                                    
    SEAL_SEPARATE_STATES.Fault :
END_CASE


CASE releaseAndFeedSubState OF
    RELEASE_FEED_STATES.Idle :                        //
                                                        
    RELEASE_FEED_STATES.MoveJawOutAndDropBag :        // 
                                                    IF (motorizedSealFlatteners.state = SEAL_FLATTENER_STATES.MovedFlattenersOut OR NOT motorizedSealFlatteners.enable) 
                                                        AND (pressureBar.clamped OR NOT pressureBar.enable)
                                                        AND ((bagDelivery.state = BAG_DELIVERY_STATES.ReverseDone) OR Globals.enableDryCycle)
                                                        OR (bagDelivery.state =  BAG_DELIVERY_STATES.WaitingForPrinter AND zebraPrinter.enable)
                                                        OR NOT bagDelivery.enable
                                                        THEN
                                                            IF motorizedSealFlatteners.enable THEN
                                                                motorizedSealFlatteners.AutoMoveToClearance();
                                                            END_IF
                                                            
                                                            IF enableBagOpen THEN
                                                                pressureBar.OpenJawForBagFeed();
															ELSE
																pressureBar.OpenJaw();
                                                            END_IF
                                                            //IBD.OpenFull();
// 															IF enableBagOpen THEN
// 																bagOpenFingers.Release();
// 															END_IF
															
															IF enableIBDEject THEN
																IBD.CloseIBD();
															END_IF
															
															IF enableLoadPlate THEN
																rearLoadPlateRetract.Trigger();
															END_IF
															
															IF TO_DINT(HMIData.exitConveyorDwell) <> 0 THEN
																exitConveyorRun.Trigger();
															END_IF
															
															IF TO_DINT(HMIData.externalExitConveyorDwell) <> 0 THEN
																externalExitConveyorRun.Trigger();
															END_IF
															
															IF enableLabelSideUp THEN
																forwardLoadPlateRetract.Trigger();
																loadShelfExtend.Trigger();
															END_IF
															
															IF HMIData.lpaBagEjectAssistEnable THEN
																LPA.ManualOn();
															END_IF
															IBD.OpenFull();
                                                           bagDropTimer.IN := TRUE;
														   releaseAndFeedSubState := RELEASE_FEED_STATES.MovingJawOutAndDroppingBag;
                                                    END_IF
													
	 RELEASE_FEED_STATES.MovingJawOutAndDroppingBag :
														 // If printer is enabled then perform printer operation of bag delivery, otherwise just feed new bag out.
                                                            // In the case that bagDelivery is disabled then we're done with release and feed
														IF enableBagOpen AND pressureBar.actualPosition >= 0.5 THEN
 															bagOpenFingers.Release();
 														END_IF	
														
                                                        IF bagDropTimer.Q 
															AND (motorizedSealFlatteners.state = SEAL_FLATTENER_STATES.MovedFlattenersToBagFeed OR NOT motorizedSealFlatteners.enable)
															THEN   
															bagDropTimer.IN := FALSE;
															
															IF bagDelivery.enable AND NOT zebraPrinter.enable THEN
                                                                bagDelivery.AutoFeedBagOut();
																LPA.ManualOff();
																IF HMIData.lpaDuringBagFeedEnable THEN
																	LPA.ManualOn();
																END_IF
                                                                releaseAndFeedSubState := RELEASE_FEED_STATES.MovingJawOutAndFeedingBag;
                                                            ELSIF bagDelivery.enable AND zebraPrinter.enable THEN
                                                                bagDelivery.AutoWaitForPrinter();
																LPA.ManualOff();
                                                                releaseAndFeedSubState := RELEASE_FEED_STATES.WaitForPrinter;
                                                            ELSE 
                                                                releaseAndFeedSubState := RELEASE_FEED_STATES.Done;
                                                            END_IF
                                                            (*{warning 'TODO: This is a hack to use HPA as LPA'}
														    HPA.DwellSetting := 500;		// Get rid on this - ha
													        HPA.Trigger();*)												
    													END_IF
														
    RELEASE_FEED_STATES.WaitForPrinter :            // Data Ready means the printer has a label and we're all set to print
                                                    IF zebraPrinter.state = PRINTER_STATES.DataReady THEN
                                                        releaseAndFeedSubState := RELEASE_FEED_STATES.FeedToOffset;
                                                    END_IF
                                                    
    RELEASE_FEED_STATES.FeedToOffset :              // This starts feeding to the print offset
													IF (motorizedSealFlatteners.state = SEAL_FLATTENER_STATES.MovedFlattenersToBagFeed OR NOT motorizedSealFlatteners.enable) THEN
														bagDelivery.AutoPrinterReady();
                                                    	releaseAndFeedSubState := RELEASE_FEED_STATES.FeedingToOffset;
													END_IF
                                                    
                                                        
    RELEASE_FEED_STATES.FeedingToOffset :            // Once offset done start printing
                                                    IF bagDelivery.state = BAG_DELIVERY_STATES.FedToPrintOffset THEN
                                                        releaseAndFeedSubState := RELEASE_FEED_STATES.StartPrinting;
                                                    END_IF                                            
    
    RELEASE_FEED_STATES.StartPrinting :                // Printer starts print cycle and bag delivery starts moving at print speed
                                                    
                                                    //bagDelivery.AutoStartPrintFeed();
													zebraPrinter.AutoPrintNow();
                                                    
                                                    releaseAndFeedSubState := RELEASE_FEED_STATES.SendPrintSignal;                                            

    RELEASE_FEED_STATES.SendPrintSignal:            // 
                                                    //IF bagDelivery.state =     BAG_DELIVERY_STATES.FeedingAtPrintSpeed THEN
													//zebraPrinter.AutoSendPrintSignal();
													IF zebraPrinter.printHeadDebounced THEN
														bagDelivery.AutoStartPrintFeed();
														zebraPrinter.AutoSendPrintSignal();
														barcodeVerifier.Trigger();
                                                        //bagDelivery.AutoStartPrintFeed();
														//bagDelivery.AutoStartPrintFeed();
                                                        //zebraPrinter.AutoSendPrintSignal();
														
                                                        releaseAndFeedSubState := RELEASE_FEED_STATES.Printing;
                                                    END_IF                                        

    RELEASE_FEED_STATES.Printing :                // 
													
                                                    IF zebraPrinter.state = PRINTER_STATES.DonePrinting THEN
                                                        releaseAndFeedSubState := RELEASE_FEED_STATES.StopPrinting;
                                                    END_IF
                                                    
    RELEASE_FEED_STATES.StopPrinting :                // Tell bag delivery it's okay to feed out the rest of the bag and the printer that it can prep itself for the next print
                                                    bagDelivery.AutoPrinterDone();
                                                    zebraPrinter.AutoAckPrintDone();
													IF HMIData.lpaDuringBagFeedEnable THEN
														LPA.ManualOn();
													END_IF
													
                                                    releaseAndFeedSubState := RELEASE_FEED_STATES.MovingJawOutAndFeedingBag;
                                                                                
                                                                                                            
    RELEASE_FEED_STATES.MovingJawOutAndFeedingBag :    // 
    
													
													IF (bagdelivery.state = BAG_DELIVERY_STATES.Ready OR NOT bagdelivery.enable)
                                                        AND (motorizedSealFlatteners.state = SEAL_FLATTENER_STATES.MovedFlattenersToBagFeed OR NOT motorizedSealFlatteners.enable) 
                                                        AND (pressureBar.pressureBarOpen OR NOT pressureBar.enable)
                                                        THEN
															IF LPA.DwellSetting = 0 THEN
																LPA.ManualOff();
															END_IF
															//IBD.OpenIBD();
                                                            releaseAndFeedSubState := RELEASE_FEED_STATES.MovedJawOutAndFedBag;
                                                    END_IF
                                                    
    RELEASE_FEED_STATES.MovedJawOutAndFedBag :      // Wait until bag is fed out before triggering barcode fail.
													IF barcodeVerifier.barcodeFault THEN
														barcodeVerificationFailed.Trigger();
													END_IF 
													
													IF enableIBDDeflate OR enableIBDEject THEN
														IBD.OpenIBD();
													END_IF
													releaseAndFeedSubState := RELEASE_FEED_STATES.Done;
    RELEASE_FEED_STATES.Done :
    RELEASE_FEED_STATES.Fault :
END_CASE

CASE openBagSubState OF
    BAG_OPEN_ASSIST_STATES.Idle :                    // 
                                                    
                                                    
                                                    
    BAG_OPEN_ASSIST_STATES.MoveJawIn :                // Close jaw against bag. In the future we may also start vacuum here
                                                    pressureBar.CloseJawNoLatch();
													(*HPA.DwellSetting := 80;
													HPA.Trigger();*)
													IF HPA.DwellSetting <> 0 THEN
														HPA.Trigger();	
													END_IF
													
													//oVacOn := TRUE; // Hard coded for now, this is vacuum
                                                    openBagSubState := BAG_OPEN_ASSIST_STATES.MovingJawIn;        
                                                    
                                                    
    BAG_OPEN_ASSIST_STATES.MovingJawIn :            // Move on once jaw is closed
                                                    IF pressureBar.iPressureBarClosed OR NOT pressureBar.enable THEN
                                                        openBagSubState := BAG_OPEN_ASSIST_STATES.MovedJawIn;        
                                                    END_IF
                                                    
                                                    
    BAG_OPEN_ASSIST_STATES.MovedJawIn :                // Hold onto the bag with vacuum to build suction
                                                    vacuumHoldTimer.IN := TRUE;
													oVacOn := TRUE; // Hard coded for now, this is vacuum
													IF vacuumHoldTimer.Q THEN
														openBagSubState := BAG_OPEN_ASSIST_STATES.MoveJawOut; 
														vacuumHoldTimer.IN := FALSE;
													END_IF
                                                                   
                                                    
                                                    
    BAG_OPEN_ASSIST_STATES.MoveJawOut :                // Open the jaw and move seal flatteners in and to bag holding
                                                    pressureBar.OpenJaw();
													motorizedSealFlatteners.AutoMoveIn();
                                                    openBagSubState := BAG_OPEN_ASSIST_STATES.MovingJawOutAndGrab;
                                                    
                                                    
    BAG_OPEN_ASSIST_STATES.MovingJawOutAndGrab :    // Once everything that is enabled is homed finish cycle 
													bagOpenFingerDelay.IN := TRUE;
													IF bagOpenFingerDelay.Q THEN
														bagOpenFingers.Grab();
														bagOpenFingerDelay.IN := FALSE;

														openBagSubState := BAG_OPEN_ASSIST_STATES.CheckForSuccessfulBagGrab;
													END_IF
													  

	BAG_OPEN_ASSIST_STATES.CheckForSuccessfulBagGrab : 	//
														IF bagOpenRetryCount < bagOpenRetrySetting THEN
															bagOpenCheckDelay.IN := TRUE;
															IF bagOpenCheckDelay.Q THEN
																IF bagOpenFingers.CheckIfBagGrabbed(TRUE) THEN // This method checks to see if the bag is grabbed and returns true if so.
																	openBagSubState := BAG_OPEN_ASSIST_STATES.BagOpened;
																	motorizedSealFlatteners.AutoMoveIn();
																ELSE 
																	openBagSubState := BAG_OPEN_ASSIST_STATES.BagFailedToOpen;
																END_IF
																bagOpenCheckDelay.IN := FALSE;
															END_IF
														ELSE 
															motorizedSealFlatteners.AutoMoveToBagHolding();
															openBagSubState := BAG_OPEN_ASSIST_STATES.MovingJawOutAfterGrab;
														END_IF
													  
	BAG_OPEN_ASSIST_STATES.BagFailedToOpen :			// 
														bagOpenFingers.Release();
														bagOpenRetryCount := bagOpenRetryCount + 1;
														IF bagOpenRetryCount < bagOpenRetrySetting THEN
															openBagSubState := BAG_OPEN_ASSIST_STATES.MoveJawIn;
														ELSIF HMIData.bagOpenFeedNewBagCount < HMIData.bagOpenFeedNewBagSetting THEN
															HMIData.bagOpenFeedNewBagCount := HMIData.bagOpenFeedNewBagCount + 1;
															bagOpenRetryCount := 0;
															motorizedSealFlatteners.AutoMoveOut();
															oVacOn := FALSE;
															openBagSubState := BAG_OPEN_ASSIST_STATES.FeedNewBag;
															
														ELSE 
															//IF (motorizedSealFlatteners.state = SEAL_FLATTENER_STATES.Idle OR NOT motorizedSealFlatteners.enable) THEN
																motorizedSealFlatteners.AutoMoveToBagHolding();
																bagFailedToOpen.Trigger();
																
																openBagSubState := BAG_OPEN_ASSIST_STATES.MovingJawOutAfterGrab;
																bagOpenRetryCount := 0; 
																HMIData.bagOpenFeedNewBagCount := 0;
																HMIData.bagsRejectedTotal.Increment();
																Globals.rejectedBagCount := Globals.rejectedBagCount + 1;
															//END_IF
															
														END_IF
	
	BAG_OPEN_ASSIST_STATES.BagOpened :					//
														bagOpened := TRUE;
                                                    	motorizedSealFlatteners.AutoMoveToBagHolding();
														bagOpenRetryCount := 0;
														HMIData.bagOpenFeedNewBagCount := 0;
														
														openBagSubState := BAG_OPEN_ASSIST_STATES.MovingJawOutAfterGrab; 
														
                                      
    BAG_OPEN_ASSIST_STATES.MovingJawOutAfterGrab :		// 
														IF (pressureBar.pressureBarOpen OR NOT pressureBar.enable) 
															AND (motorizedSealFlatteners.state = SEAL_FLATTENER_STATES.Idle OR NOT motorizedSealFlatteners.enable)
															THEN
																openBagSubState := BAG_OPEN_ASSIST_STATES.MovedJawOut;        
														END_IF	 
														
	
	BAG_OPEN_ASSIST_STATES.MovedJawOut :            // 
														oVacOn := FALSE; 		// Hard coded for now, this is vacuum
														
														
														openBagSubState := BAG_OPEN_ASSIST_STATES.Done;

                                                             
                                                
	BAG_OPEN_ASSIST_STATES.FeedNewBag :   			//
													IF (motorizedSealFlatteners.state = SEAL_FLATTENER_STATES.Idle OR NOT motorizedSealFlatteners.enable) THEN
														state := HEAD_STATES.SealAndSeparateBag;
													END_IF
													
													
                                                
    BAG_OPEN_ASSIST_STATES.Done :                    // 
                                                            
    BAG_OPEN_ASSIST_STATES.Fault :                    //
													

END_CASE

CASE finishCycleSubState OF
	FINISH_CYCLE_STATES.Idle:								//
	
	FINISH_CYCLE_STATES.Start :								//
															IF funnel.enable THEN
																finishCycleSubState := FINISH_CYCLE_STATES.OpenFunnel;
															ELSIF enableBagOpen THEN
																finishCycleSubState := FINISH_CYCLE_STATES.Done;
															ELSE
																IF motorizedSealFlatteners.enable THEN
																	finishCycleSubState := FINISH_CYCLE_STATES.BringSealFlattenersInAndDown;
																ELSE
																	finishCycleSubState := FINISH_CYCLE_STATES.Done;
																END_IF
															END_IF
															IF LPA.DwellSetting <> 0 THEN
																LPA.Trigger();
															END_IF
	
	FINISH_CYCLE_STATES.OpenFunnel :						//
															IF LPA.DwellSetting <> 0 THEN
																LPA.Trigger();
															END_IF
															funnel.OpenNow();
															finishCycleSubState := FINISH_CYCLE_STATES.OpeningFunnel;
	
	FINISH_CYCLE_STATES.OpeningFunnel :						//
															IF funnel.opened THEN
																finishCycleSubState := FINISH_CYCLE_STATES.OpenedFunnel;
															END_IF
	
	FINISH_CYCLE_STATES.OpenedFunnel :						//
															//IF enableBagOpen THEN
																IF iLefttFingerBagPresent AND iRightFingerBagPresent THEN
																	finishCycleSubState := FINISH_CYCLE_STATES.Done;
																ELSE
																	IF bagOpenRetryCount < bagOpenRetrySetting THEN
																		bagOpenRetryCount := bagOpenRetryCount + 1;
																		funnel.CloseNow();
																		finishCycleSubState := FINISH_CYCLE_STATES.ClosingFunnelForRetry;
																	ELSE
																		bagFailedToOpen.Trigger();
																		funnel.CloseNow();
																		bagOpenRetryCount := 0; 
																		HMIData.bagsRejectedTotal.Increment();
																		finishCycleSubState := FINISH_CYCLE_STATES.Done;
																	END_IF
																END_IF
															ELSE
																IF motorizedSealFlatteners.enable THEN
																	finishCycleSubState := FINISH_CYCLE_STATES.BringSealFlattenersToBagHolding;
																ELSE
																	finishCycleSubState := FINISH_CYCLE_STATES.Done;
																END_IF
															//END_IF
	
	FINISH_CYCLE_STATES.ClosingFunnelForRetry :				//
															IF funnel.closed THEN
																finishCycleSubState := FINISH_CYCLE_STATES.Start;
															END_IF												
	
	FINISH_CYCLE_STATES.BringSealFlattenersInAndDown :		//
															motorizedSealFlatteners.AutoMoveToHandLoad();
															finishCycleSubState := FINISH_CYCLE_STATES.BringingSealFlattenersInAndDown;
	
	FINISH_CYCLE_STATES.BringingSealFlattenersInAndDown :	//
															IF motorizedSealFlatteners.state = SEAL_FLATTENER_STATES.Idle THEN
																finishCycleSubState := FINISH_CYCLE_STATES.SealFlattenersInAndDown;
															END_IF
	
	FINISH_CYCLE_STATES.SealFlattenersInAndDown :			//
															finishCycleSubState := FINISH_CYCLE_STATES.Done;
	
	FINISH_CYCLE_STATES.BringSealFlattenersToBagHolding:	//
															motorizedSealFlatteners.AutoMoveToBagHolding();
															finishCycleSubState := FINISH_CYCLE_STATES.BringingSealFlattenersToBagHolding;
	
	FINISH_CYCLE_STATES.BringingSealFlattenersToBagHolding: //
															IF motorizedSealFlatteners.state = SEAL_FLATTENER_STATES.Idle THEN
																finishCycleSubState := FINISH_CYCLE_STATES.SealFlattenersAtBagHolding;
															END_IF
																
	FINISH_CYCLE_STATES.SealFlattenersAtBagHolding : 		//
															finishCycleSubState := FINISH_CYCLE_STATES.Done;
	
	FINISH_CYCLE_STATES.Done :								//
															bagOpenRetryCount := 0;
														
	
	FINISH_CYCLE_STATES.Fault :
	
	
END_CASE
HMIData.initiateCycle := FALSE;

END_FUNCTION_BLOCK

// FBs/Components/FB_MotorizedPressureBar/FB_MotorizedPressureBar
FUNCTION_BLOCK FB_MotorizedPressureBar EXTENDS BaseComponentFB
VAR_INPUT
	iPressureBarClamped: BOOL;
	iPressureBarClosed : BOOL;
	iPressureBarNotObstructed : BOOL;
	iBaggerEnableButton : BOOL;
	iJawClampExtended : BOOL;
	iJawCLampRetracted : BOOL;
	pbarOutSetting : REAL := 12.0;
	pbarBagFeedSetting : REAL := 2.0;
	pbarInSetting : REAL := 0.0;
	closeDelay : REAL;
	disableFaults : BOOL;
	extendJawClamp : BOOL;
	retractJawClamp : BOOL;
	extendJaw : BOOL;
	retractJaw : BOOL;
END_VAR
VAR_OUTPUT
	
	
	failToClampLeft : FB_Fault(name := 'Pbar Left Fail to Clamp');
	failToReleaseLeft : FB_Fault(name := 'Pbar Left Fail to Release');
	failToClampRight : FB_Fault(name := 'Pbar Right Fail to Clamp');
	failToReleaseRight : FB_Fault(name := 'Pbar Right Fail to Release');
	faults : PressureBarFaultsType;
	state : MotorizedPbarStates;
	actualPosition : REAL;
	pressureBarOpen : BOOL;
	pressureBarClosed : BOOL;
	homeRequired : BOOL;
	clamped : BOOL;
END_VAR
VAR
	_homeNow : BOOL;
	_openJaw : BOOL;
	_closeJaw : BOOL;
	_closeJawNoLatch : BOOL;
	_openForBagFeed : BOOL;
	jawClampsDelay : TIME := T#75MS;
	accel : INT := 150;
	decel : INT := 100;
	velo : INT := 1250;
	testCurrent : DINT := 500;
	testZeroCurrent : BOOL;
	testSomeCurrent : BOOL;
	testClamp : BOOL;
	testRelease : BOOL;
	testPosLimit : BOOL;
	testDisable : BOOL;
	testEnable : BOOL;
	testResetPosition : BOOL;
	posLimit : DINT := 3000;
	pbarFeedbackHandler : FB_CylinderFeedback;
	jawClampsLeftFeedbackHandler : FB_CylinderFeedback;
	jawClampsRightFeedbackHandler : FB_CylinderFeedback;
	startTest : BOOL;
	testActive : BOOL;
	movePassthroughNow : BOOL;
	delayTimer : Standard.TON := (PT:= T#500MS);
	failTimer : Standard.TON := (PT:= T#500MS);
	homeRequiredONS : FB_ONS;
	faultingONS : FB_ONS;
	faultTimeMultiplier : REAL := 150;
	distanceToMove : REAL;
	disableMotorONS : FB_ONS;
	pbarOutCommandedSetting : REAL;
	strokeTimer : Standard.TON;
	strokeTime : TIME;
	movingONS : FB_ONS;
END_VAR
VAR_IN_OUT
	jawClamps : FB_ThreePositionCylinder;
	pbarMotor : FB_AppliedMotionStepServoEIPPassthrough;
	//IBDMotor : FB_AppliedMotionStepServoEIPPassthrough;
END_VAR


actualPosition := pbarMotor.absolutePositonInches;
pressureBarOpen := TO_DINT(actualPosition * 1000) >= (TO_DINT(pbarOutCommandedSetting * 1000) - 10) AND TO_DINT(actualPosition * 1000) <= (TO_DINT(pbarOutCommandedSetting * 1000) + 10);
//pressureBarClosed := pbarMotor.absolutePositionSteps >= (pbarMotor.distanceToMoveInSteps - 4) AND pbarMotor.absolutePositionSteps <= (pbarMotor.distanceToMoveInSteps + 4);
pressureBarClosed := iPressureBarClosed;
delayTimer();
failTimer(IN := (state = MotorizedPbarStates.StartedClamping) AND (NOT (iJawCLampRetracted AND iPressureBarClamped AND iPressureBarClosed)));
clamped := state = MotorizedPbarStates.Clamping;

strokeTimer();
movingONS(CLK := state = MotorizedPbarStates.MovingJawIn);

IF movingONS.OSR THEN
	strokeTimer.IN := TRUE;
END_IF
IF movingONS.OSF THEN
	strokeTime := strokeTimer.ET;
	strokeTimer.IN := FALSE;
END_IF
	

disableMotorONS(CLK := clamped AND iPressureBarClamped AND iJawClampsRetracted);
IF disableMotorONS.OSR THEN
	pbarMotor.AllowClamping();
END_IF



// jawClampsLeftFeedbackHandler(
// 	extendedFeedbackInput:= iJawClampLeftExtended, 
// 	retractedFeedbackInput:= iJawCLampLeftRetracted, 
// 	extendOutput:= jawClamps.extendOutput, 
// 	retractOutput:= jawClamps.retractOutput, 
// 	extendFaultDelay:= 1000, 
// 	retractFaultDelay:= 1000, 
// 	faultMonitoring:= NOT disableFaults, 
// 	failedToExtend=> failToReleaseLeft.faultTrigger, 
// 	failedToRetract=> failToClampLeft.faultTrigger);
// 
// jawClampsRightFeedbackHandler(
// 	extendedFeedbackInput:= iJawClampRightExtended, 
// 	retractedFeedbackInput:= iJawCLampRightRetracted, 
// 	retractOutput:= jawClamps.retractOutput, 
// 	extendOutput:= jawClamps.extendOutput, 
// 	extendFaultDelay:= 1000, 
// 	retractFaultDelay:= 1000, 
// 	faultMonitoring:= NOT disableFaults, 
// 	failedToExtend=> failToReleaseRight.faultTrigger, 
// 	failedToRetract=> failToClampRight.faultTrigger);


IF extendJawClamp THEN
	extendJawClamp := FALSE;
	jawClamps.Extend();
ELSIF retractJawClamp THEN
	retractJawClamp := FALSE;
	jawClamps.Retract();
END_IF

IF NOT pbarMotor.HomeRequired THEN
	IF extendJaw THEN
		extendJaw := FALSE;
		pbarMotor.MoveToPositionTorque(pbarOutSetting,accel,decel,velo,testCurrent);
	ELSIF retractJaw THEN
		retractJaw := FALSE;
		pbarMotor.MoveToPositionTorque(pbarInSetting,accel,decel,velo,testCurrent);
	END_IF
END_IF

IF testDisable THEN
	pbarMotor.Disable();
	testDisable := FALSE;
END_IF

IF testEnable THEN
	pbarMotor.Enable();
	testEnable := FALSE;
END_IF

IF testClamp THEN
	pbarMotor.AllowClamping();
	testClamp := FALSE;
END_IF

IF testRelease THEN
	pbarMotor.DoneClamping();
	testRelease := FALSE;
END_IF

IF testResetPosition THEN
	pbarMotor.ResetEncoderPosition(pbarMotor.driveInputs[5]);
	testResetPosition := FALSE;
END_IF

IF testZeroCurrent THEN
	pbarMotor.MoveDistanceTorque(velocity:=100, acceleration := 1, deceleration := 1, distance := 0, current := 1);
	//pbarMotor.SetTorque(1);
	testZeroCurrent := FALSE;
END_IF

IF testSomeCurrent THEN
	pbarMotor.SetTorque(testCurrent);
	testSomeCurrent := FALSE;
END_IF

IF testPosLimit THEN
	pbarMotor.SetPositionLimit(posLimit);
	testPosLimit := FALSE;
END_IF

IF resetONS.Q THEN
	pbarMotor.Reset();
	//pbarMotor.Enable();
	pbarMotor.ResetEncoderPosition(pbarMotor.driveInputs[5]);
	//IBDMotor.Reset();
	Globals.jawMovingIn := FALSE;
	_reset := FALSE;
	startTest := FALSE;
	testActive := FALSE;
	delayTimer.IN := FALSE;
	pbarMotor.DoneClamping();
	jawClamps.Extend();
	pbarFeedbackHandler.extendOutput := FALSE;
	pbarFeedbackHandler.retractOutput := FALSE;
	state := MotorizedPbarStates.Idle; 
END_IF
faultingONS(CLK := (	pbarMotor.Faulted AND NOT disableFaults)
	OR (pbarFeedbackHandler.faultIndication
	OR jawClampsLeftFeedbackHandler.faultIndication
	OR jawClampsRightFeedbackHandler.faultIndication
	OR faults.obstructionDetected.active));

IF 	faultingONS.OSR
	AND state <> MotorizedPbarStates.Faulted 
THEN
	state := MotorizedPbarStates.Faulting; 
END_IF

homeRequiredONS(CLK := pbarMotor.homeRequired);
IF homeRequiredONS.OSR THEN
	homeRequired := TRUE;
END_IF


_ready := state = MotorizedPbarStates.Idle AND NOT homeRequired AND pressureBarOpen;

CASE state OF
	MotorizedPbarStates.Idle :					//
										IF startTest THEN
											startTest := FALSE;
											testActive := TRUE;
											IF pbarMotor.homeRequired THEN
												pbarMotor.HomeNow();
												state := MotorizedPbarStates.Homing;
											ELSE
												state := MotorizedPbarStates.Initialize;
											END_IF
												
										END_IF
											
										IF _homeNow THEN
											_homeNow := FALSE;
											//IF (pbarMotor.homeRequired) THEN
												pbarMotor.HomeNow();
											//END_IF
											delayTimer.PT := T#150MS;
											delayTimer.IN := TRUE;
											state := MotorizedPbarStates.Homing;
										END_IF
										
										IF _openJaw AND NOT _reset THEN
											//pbarMotor.DoneClamping();
											_openJaw := FALSE;
											pbarOutCommandedSetting := pbarOutSetting;
											state := MotorizedPbarStates.MoveJawOut;
										END_IF
										
										IF _openForBagFeed AND NOT _reset THEN
											//pbarMotor.DoneClamping();
											_openForBagFeed := FALSE;
											pbarOutCommandedSetting := pbarBagFeedSetting;
											state := MotorizedPbarStates.MoveJawOut;
										END_IF
										
										IF _closeJaw THEN
											_closeJaw := FALSE;
											state := MotorizedPbarStates.MoveJawIn;
										END_IF
										
										IF _closeJawNoLatch THEN
											//_closeJawNoLatch := FALSE;
											state := MotorizedPbarStates.MoveJawIn;
										END_IF
	
	MotorizedPbarStates.Homing :				//
										Globals.jawMovingIn := TRUE;
										IF NOT (pbarMotor.homeRequired) AND delayTimer.Q THEN
												delayTimer.IN := FALSE;
												//pbarMotor.DoneClamping();
												
												homeRequired := FALSE;
												
												state := MotorizedPbarStates.Initialize;
										END_IF
	
	
	MotorizedPbarStates.Initialize :			//
										delayTimer.PT := T#500MS;
										delayTimer.IN := TRUE;
										Globals.jawMovingIn := TRUE;
										IF delayTimer.Q THEN
											IF pressureBarOpen THEN
												pbarMotor.DoneClamping();
												state := MotorizedPbarStates.Initializing;
											ELSE
												jawClamps.Extend();
												pbarMotor.MoveToPositionTorque(pbarOutSetting,accel,decel,velo,testCurrent);
												//IBDMotor.MoveToPosition(pbarOutSetting,accel,decel,velo);
												state := MotorizedPbarStates.Initializing;
											END_IF
											delayTimer.IN := FALSE;
										END_IF
										
	
	
	MotorizedPbarStates.Initializing :			//
										IF pressureBarOpen THEN
											state := MotorizedPbarStates.Initialized;
										END_IF
	
	
	MotorizedPbarStates.Initialized :			//
										IF testActive THEN
											state := MotorizedPbarStates.MoveJawIn;
										ELSE
											state := MotorizedPbarStates.Idle;
										END_IF
										pbarMotor.SetPositionLimit(posLimit);
										
	
	
	MotorizedPbarStates.MoveJawOut :			//
										
										Globals.jawMovingIn := FALSE;
										pbarMotor.MoveToPositionTorque(pbarOutCommandedSetting,accel,decel,velo,testCurrent);
										//IBDMotor.MoveToPosition(pbarOutSetting,accel,decel,velo);
										distanceToMove := ABS(actualPosition - pbarOutCommandedSetting);
										state := MotorizedPbarStates.MovingJawOut;
										//pbarMotor.SetPositionLimit(150);
	
	MotorizedPbarStates.MovingJawOut :			//
										IF pressureBarOpen THEN
											
											IF testActive THEN
												delayTimer.PT := T#500MS;
												delayTimer.IN := TRUE;
												IF delayTimer.Q  THEN
													delayTimer.IN := FALSE;
													state := MotorizedPbarStates.MoveJawIn;
												END_IF
											ELSE
												delayTimer.PT := T#100MS;
												delayTimer.IN := TRUE;
												IF delayTimer.Q  THEN
													//pbarMotor.ResetEncoderPosition(pbarMotor.driveInputs[5]);
													delayTimer.IN := FALSE;
													state := MotorizedPbarStates.Idle;
												END_IF
											END_IF
										END_IF
	
	
	MotorizedPbarStates.MovedJawOut :			//
										IF delayTimer.Q THEN
											delayTimer.IN := FALSE;
											state := MotorizedPbarStates.MoveJawIn;
										END_IF
	
	
	MotorizedPbarStates.MoveJawIn :				//
										Globals.jawMovingIn := TRUE;
										pbarMotor.MoveToPositionTorque(pbarInSetting,accel,decel,velo,testCurrent);
										//pbarMotor.MoveToPositionTorque(pbarInSetting,accel,decel,velo,testCurrent);
										//IBDMotor.MoveToPosition(0,accel,decel,velo+(TO_INT(TO_REAL(velo)*0.25)));
										distanceToMove := ABS(actualPosition - pbarInSetting);
										state := MotorizedPbarStates.MovingJawIn;
	
	
	MotorizedPbarStates.MovingJawIn : 			//
										//IF iPressureBarClosed AND pbarMotor.absolutePositonInches = 0 THEN
										IF iPressureBarClosed THEN
											IF NOT  _closeJawNoLatch THEN
												//pbarMotor.AllowClamping();
											END_IF
											
											delayTimer.PT := jawClampsDelay;
											delayTimer.IN := TRUE;
											//pbarMotor.Disable();
											state := MotorizedPbarStates.MovedJawIn;
										END_IF
	
	
	MotorizedPbarStates.MovedJawIn :			//
										//IF delayTimer.Q THEN
											delayTimer.IN := FALSE;
											IF _closeJawNoLatch THEN
												_closeJawNoLatch := FALSE;
												state := MotorizedPbarStates.Idle;
											ELSE
												state := MotorizedPbarStates.StartClamping;
											END_IF
										//END_IF
										
	
	
	MotorizedPbarStates.StartClamping :			//
										//pbarMotor.SetPositionLimit(20000);
										jawClamps.Retract();
										state := MotorizedPbarStates.StartedClamping;
	
	MotorizedPbarStates.StartedClamping :		//
										IF iPressureBarClamped AND iJawClampsRetracted THEN
											
											//pbarMotor.AllowClamping();
											delayTimer.PT := T#250MS;
											delayTimer.IN := TRUE;
											IF delayTimer.Q THEN
												//pbarMotor.AllowClamping();
												pbarMotor.ResetEncoderPosition(pbarMotor.driveInputs[5]);
												state := MotorizedPbarStates.Clamping;	
											END_IF
										END_IF
										
										
										IF testActive THEN
											delayTimer.PT := T#2S;
											delayTimer.IN := TRUE;
										END_IF
	
	
	MotorizedPbarStates.Clamping :				//
										IF _openJaw OR (testActive AND delayTimer.Q) THEN
											_openJaw := FALSE;
											pbarOutCommandedSetting := pbarOutSetting;
											delayTimer.IN := FALSE;
											jawClamps.Extend();
											state := MotorizedPbarStates.ReleaseClamp;
										END_IF
										
										IF _openForBagFeed OR (testActive AND delayTimer.Q) THEN
											_openForBagFeed := FALSE;
											pbarOutCommandedSetting := pbarBagFeedSetting;
											delayTimer.IN := FALSE;
											jawClamps.Extend();
											state := MotorizedPbarStates.ReleaseClamp;
										END_IF
										
	
	
	
	MotorizedPbarStates.ReleaseClamp :			//  
										IF iJawClampExtended THEN
											pbarMotor.DoneClamping();
											//pbarMotor.Enable();
											delayTimer.PT := jawClampsDelay;
											delayTimer.IN := TRUE;
											state := MotorizedPbarStates.ReleasingClamp;
										END_IF
										
	
	
	MotorizedPbarStates.ReleasingClamp :		//
										IF delayTimer.Q THEN
											delayTimer.IN := FALSE;
											state := MotorizedPbarStates.MoveJawOut;
											//HMI.data.TFBeltPressureBarCycles := HMI.data.TFBeltPressureBarCycles + 1;
										END_IF
	
	MotorizedPbarStates.Faulting :			// 
										Globals.jawMovingIn := FALSE;
										_reset := FALSE;
										_openJaw := FALSE;
										_closeJaw := FALSE;
										_homeNow := FALSE;
										_closeJawNoLatch := FALSE;
										_openForBagFeed := FALSE;
										startTest := FALSE;
										testActive := FALSE;
										delayTimer.IN := FALSE;
										jawClamps.Extend();
										pbarFeedbackHandler.extendOutput := FALSE;
										pbarFeedbackHandler.retractOutput := FALSE;
										pbarMotor.Disable();
										//IBDMotor.Disable();
										state := MotorizedPbarStates.Faulted;
			
	MotorizedPbarStates.Faulted :				//
	
END_CASE


IF pbarMotor.alarms.positionLimit OR failTimer.Q THEN
	faults.obstructionDetected.faultTrigger := TRUE;
	//homeRequired := TRUE;
	//state := MotorizedPbarStates.Faulting;
ELSE
	faults.obstructionDetected.faultTrigger := FALSE;
END_IF

pbarFeedbackHandler(
	extendedFeedbackInput:= pressureBarOpen, 
	retractedFeedbackInput:= iPressureBarClosed, 
	extendOutput:= state = MotorizedPbarStates.MovingJawOut, 
	retractOutput:= state = MotorizedPbarStates.MovingJawIn, 
	extendFaultDelay:= 3000 , 
	retractFaultDelay:= 3000 , 
	faultMonitoring:= distanceToMove > 0.5, 
	failedToExtend=> faults.failedToOpen.faultTrigger, 
	failedToRetract=> faults.failedToClose.faultTrigger);
	
SUPER^();

METHOD CloseJawNoLatch : BOOL
VAR_INPUT
END_VAR
_closeJawNoLatch := TRUE;
END_METHOD

METHOD OpenJaw : BOOL
VAR_INPUT
END_VAR
_openJaw := TRUE;
END_METHOD

METHOD CloseJaw : BOOL
VAR_INPUT
END_VAR
_closeJaw := TRUE;
END_METHOD

METHOD OpenJawForBagFeed : BOOL
VAR_INPUT
END_VAR
_openForBagFeed := TRUE;
END_METHOD

METHOD HomeNow : BOOL
VAR_INPUT
END_VAR
_homeNow := TRUE;
END_METHOD

END_FUNCTION_BLOCK

// FBs/Components/FB_MotorizedPressureBar/FB_CylinderFeedback
FUNCTION_BLOCK FB_CylinderFeedback
VAR_INPUT
    extendedFeedbackInput : BOOL;    //Extended feedback input from I/O
    retractedFeedbackInput : BOOL;    //Retracted feedback input from I/O
	extendOutput : BOOL;				// Extend output from valve
	retractOutput : BOOL; 				// Retract output from valve
    extendFaultDelay : INT := 1000;        //Extend fault delay in MS
    retractFaultDelay : INT := 1000;        //Retract fault delay in MS
    faultMonitoring : BOOL;                    //Fault monitoring enabled if true
END_VAR
VAR_OUTPUT
    failedToExtend : BOOL;            //Failed to Extend Fault
    failedToRetract : BOOL;            //Failed to Retract Fault
	faultIndication : BOOL;            //Overall fault status of cylinder
END_VAR
VAR
    
    extendFaultTimer : TON;            //Extend Fault Timer
    retractFaultTimer : TON;        //Retract Fault Timer
END_VAR

//This code monitors the positon of the cylinder and raises a fault if the cylinder doesn't reach its
//desired postion within the specified time.

//Initialize timers
extendFaultTimer(PT := INT_TO_TIME(extendFaultDelay));
retractFaultTimer(PT := INT_TO_TIME(retractFaultDelay));

//Only enable timers if we are to be monitoring faults
IF faultMonitoring THEN
    extendFaultTimer.IN := (extendOutput AND NOT extendedFeedbackInput);
    retractFaultTimer.IN := (retractOutput AND NOT retractedFeedbackInput);
ELSE 
        extendFaultTimer.IN := FALSE;
        retractFaultTimer.IN := FALSE;
END_IF

//Rasie the alarms
failedToExtend := extendFaultTimer.Q;
failedToRetract := retractFaultTimer.Q;

//Set overall fault indication
faultIndication := failedToExtend OR failedToRetract;

END_FUNCTION_BLOCK

// FBs/Components/FB_MotorizedIBD/FB_MotorizedIBD
FUNCTION_BLOCK FB_MotorizedIBD EXTENDS BaseComponentFB
VAR_INPUT
	pbarOutSetting : REAL := 12.0;
	IBDOutCalculated : REAL := 12.0;
	pbarInSetting : REAL;
	IBDOffset : REAL := 2.0;
	disableFaults : BOOL;
	extendCommand : BOOL;
	retractCommand : BOOL;
END_VAR
VAR_OUTPUT
	failToOpen : FB_Fault(name := 'IBD Fail to Open');
	state : MotorizedIBDStates;
	actualPosition : REAL;
	IBDOpen : BOOL;
	IBDFullyOpen : BOOL;
	homeRequired : BOOL;
	clamped : BOOL;
END_VAR
VAR
	_homeNow : BOOL;
	_openIBD : BOOL;
	_closeIBD : BOOL;
	_openFull : BOOL;
	accel : INT := 150;
	decel : INT := 100;
	velo : INT := 1250;
	testCurrent : DINT := 500;
	testZeroCurrent : BOOL;
	testSomeCurrent : BOOL;
	startTest : BOOL;
	testActive : BOOL;
	movePassthroughNow : BOOL;
	delayTimer : Standard.TON := (PT:= T#500MS);
	failToOpenTimer : Standard.TON := (PT := T#2s);
	homeRequiredONS : FB_ONS;
	faultingONS : FB_ONS;
END_VAR
VAR_IN_OUT
	IBDMotor : FB_AppliedMotionStepServoEIPPassthrough;
END_VAR


actualPosition := IBDMotor.absolutePositonInches;
IBDOpen := TO_DINT(actualPosition * 1000) >= (TO_DINT((pbarOutSetting) * 1000) - 10) AND TO_DINT(actualPosition * 1000) <= (TO_DINT((pbarOutSetting)* 1000) + 10);
IBDFullyOpen := TO_DINT(actualPosition * 1000) >= (TO_DINT(12 * 1000) - 10) AND TO_DINT(actualPosition * 1000) <= (TO_DINT(12 * 1000) + 10);
//IBDOpen := TO_DINT(IBDMotor.absolutePositonInches) = TO_DINT(pbarOutSetting);
delayTimer();

clamped := state = MotorizedIBDStates.Clamping;

failToOpenTimer(IN := state = MotorizedIBDStates.MovingJawOut OR state = MotorizedIBDStates.MovingOutFull);

IF NOT IBDMotor.HomeRequired THEN
	IF extendCommand THEN
		extendCommand := FALSE;
		IBDMotor.MoveToPositionTorque(pbarOutSetting,accel,decel,velo,testCurrent);
	ELSIF retractCommand THEN
		retractCommand := FALSE;
		IBDMotor.MoveToPositionTorque(pbarInSetting,accel,decel,velo,testCurrent);
	END_IF
END_IF


IF testZeroCurrent THEN
	IBDMotor.SetTorque(0);
	testZeroCurrent := FALSE;
END_IF

IF testSomeCurrent THEN
	IBDMotor.SetTorque(testCurrent);
	testSomeCurrent := FALSE;
END_IF


IF resetONS.Q THEN
	//IF IBDMotor.Faulted THEN
		IBDMotor.Reset();
	//END_IF
	IBDMotor.ResetEncoderPosition(IBDMotor.driveInputs[5]);
	_reset := FALSE;
	_openIBD := FALSE;
	_closeIBD := FALSE;
	_homeNow := FALSE;
	startTest := FALSE;
	testActive := FALSE;
	delayTimer.IN := FALSE;
	state := MotorizedIBDStates.Idle; 
END_IF
faultingONS(CLK := IBDMotor.Faulted AND NOT disableFaults);

IF (faultingONS.OSR AND disableFaults)
	AND state <> MotorizedIBDStates.Faulted
THEN
	state := MotorizedIBDStates.Faulting; 
END_IF

homeRequiredONS(CLK := IBDMotor.homeRequired);
IF homeRequiredONS.OSR THEN
	homeRequired := TRUE;
END_IF

_ready := state = MotorizedIBDStates.Idle AND NOT homeRequired AND IBDOpen;

CASE state OF
	MotorizedIBDStates.Idle :					//
										IF startTest THEN
											startTest := FALSE;
											testActive := TRUE;
											IF IBDMotor.homeRequired THEN
												IBDMotor.HomeNow();
												state := MotorizedIBDStates.Homing;
											ELSE
												state := MotorizedIBDStates.Initialize;
											END_IF
												
										END_IF
											
										
										IF IBDMotor.status.motorEnabled THEN
											IF _openIBD AND NOT _reset THEN
											_openIBD := FALSE;
											state := MotorizedIBDStates.MoveJawOut;
										END_IF
										
										IF _closeIBD THEN
											_closeIBD := FALSE;
											state := MotorizedIBDStates.MoveJawIn;
										END_IF
										
										IF _openFull THEN
											_openFull := FALSE;
											state := MotorizedIBDStates.MoveOutFull;
										END_IF
										
										IF _homeNow THEN
											_homeNow := FALSE;
											//IF IBDMotor.HomeRequired THEN
												IBDMotor.HomeNow();
											//END_IF
											delayTimer.PT := T#150MS;
											delayTimer.IN := TRUE;
											state := MotorizedIBDStates.Homing;
										END_IF
										END_IF
										
	
	MotorizedIBDStates.Homing :				//
										
										IF NOT (IBDMotor.homeRequired) AND delayTimer.Q THEN
											delayTimer.IN := FALSE;
											homeRequired := FALSE;
											state := MotorizedIBDStates.Initialize;
										END_IF
	
	
	MotorizedIBDStates.Initialize :			//
										
										IF IBDOpen THEN
											state := MotorizedIBDStates.Initialized;
										ELSE
											IBDMotor.MoveToPosition(pbarOutSetting,accel,decel,velo);
											//IBDMotor.MoveToPosition(pbarOutSetting,accel,decel,velo);
											state := MotorizedIBDStates.Initializing;
										END_IF
	
	
	MotorizedIBDStates.Initializing :			//
										IF IBDOpen THEN
											state := MotorizedIBDStates.Initialized;
										END_IF
	
	
	MotorizedIBDStates.Initialized :			//
										state := MotorizedIBDStates.Idle;
	
	
	MotorizedIBDStates.MoveJawOut :			//
										
										//IBDMotor.MoveToPositionTorque(pbarOutSetting,accel,decel,velo,testCurrent);
										IBDMotor.MoveToPosition(pbarOutSetting,accel,decel,velo);
										state := MotorizedIBDStates.MovingJawOut;
										_openIBD := FALSE;
										//IBDMotor.SetPositionLimit(150);
	
	MotorizedIBDStates.MovingJawOut :			//
										IF IBDOpen THEN
											state := MotorizedIBDStates.Idle;
										END_IF
	
	
	MotorizedIBDStates.MovedJawOut :			//
										
	
	MotorizedIBDStates.MoveOutFull :			//
										
										//IBDMotor.MoveToPositionTorque(pbarOutSetting,accel,decel,velo,testCurrent);
										IBDMotor.MoveToPosition(pbarOutSetting,accel,decel,velo);
										state := MotorizedIBDStates.MovingOutFull;
										//IBDMotor.SetPositionLimit(150);
	
	MotorizedIBDStates.MovingOutFull :			//
										IF IBDOpen THEN
											state := MotorizedIBDStates.Idle;
										END_IF
	
	
	MotorizedIBDStates.MovedOutFull :			//
	
	MotorizedIBDStates.MoveJawIn :				//
									
										IBDMotor.MoveToPositionTorque(pbarInSetting,accel,decel,velo,testCurrent);
										//IBDMotor.MoveToPosition(0,accel,decel,velo+(TO_INT(TO_REAL(velo)*0.25)));
										state := MotorizedIBDStates.MovingJawIn;
	
	
	MotorizedIBDStates.MovingJawIn : 			//
										IF IBDMotor.alarms.currentFoldback OR IBDMotor.InPosition THEN
											state := MotorizedIBDStates.Clamping;
										END_IF
	
	
	MotorizedIBDStates.MovedJawIn :			//
										state := MotorizedIBDStates.StartClamping;
	
	
	MotorizedIBDStates.StartClamping :			//
										
	
	MotorizedIBDStates.StartedClamping :		//
										
	
	
	MotorizedIBDStates.Clamping :				//
										IF _openIBD THEN
											_openIBD := FALSE;
											state := MotorizedIBDStates.MoveJawOut;
										END_IF
											
										IF _openFull THEN
											_openFull := FALSE;
											state := MotorizedIBDStates.MoveOutFull;
										END_IF
	
	
	MotorizedIBDStates.ReleaseClamp :			//  
										
	
	MotorizedIBDStates.ReleasingClamp :		//
										
	
	MotorizedIBDStates.Faulting :			// 
										Globals.jawMovingIn := FALSE;
										_reset := FALSE;
										_openIBD := FALSE;
										_closeIBD := FALSE;
										_homeNow := FALSE;
										startTest := FALSE;
										testActive := FALSE;
										delayTimer.IN := FALSE;
										//IBDMotor.MoveDistanceTorque(velocity:=100, acceleration := 1, deceleration := 1, distance := 0, current := 0);
										IBDMotor.Disable();
										state := MotorizedIBDStates.Faulted;
	
	MotorizedIBDStates.Faulted :				//
	
END_CASE

SUPER^();

METHOD CloseIBD : BOOL
VAR_INPUT
END_VAR
_closeIBD := TRUE;
END_METHOD

METHOD OpenFull : BOOL
VAR_INPUT
END_VAR
_openFull := TRUE;
END_METHOD

METHOD OpenIBD : BOOL
VAR_INPUT
END_VAR
_openIBD := TRUE;
END_METHOD

METHOD RemovePower : BOOL
VAR_INPUT
END_VAR
state := MotorizedIBDStates.Faulting;
//homeRequired := TRUE;
END_METHOD

METHOD HomeNow : BOOL
VAR_INPUT
END_VAR
_homeNow := TRUE;
END_METHOD

END_FUNCTION_BLOCK

// FBs/FB_BaggerHeadRaise
FUNCTION_BLOCK FB_BaggerHeadRaise
VAR_INPUT
	faultIndication : BOOL;
	raiseCommand : BOOL;
	lowerCommand : BOOL;
	raiseLimitSwitch : BOOL;
	lowerLimitSwitch : BOOL;
END_VAR
VAR_OUTPUT
	runMotorOutput : BOOL;
	motorDirectionOutput : BOOL;
END_VAR
VAR
END_VAR

IF NOT faultIndication THEN
	IF (raiseCommand AND NOT raiseLimitSwitch) OR (lowerCommand AND NOT lowerLimitSwitch) THEN
		runMotorOutput := TRUE;
	ELSE
		runMotorOutput := FALSE;
	END_IF
	
	IF (lowerCommand AND NOT lowerLimitSwitch) THEN
		motorDirectionOutput := TRUE;
	ELSE
		motorDirectionOutput := FALSE;
	END_IF
	
ELSE
	runMotorOutput := FALSE;
	motorDirectionOutput := FALSE;
END_IF

END_FUNCTION_BLOCK

// FBs/Components/FB_MurrK50/FB_MurrK50
FUNCTION_BLOCK FB_MurrK50
VAR_INPUT
	baggerReady : BOOL;
	baggerFaulted : BOOL;
	baggerInCycle : BOOL;
END_VAR
VAR_OUTPUT
	IOLinkStateOutput : BYTE;
END_VAR
VAR
END_VAR

IOLinkStateOutput := 0;
IF baggerReady THEN
	IOLinkStateOutput := 1;
END_IF
IF baggerInCycle THEN
	IOLinkStateOutput := 2;
END_IF
IF baggerFaulted THEN
	IOLinkStateOutput := 3;
END_IF

END_FUNCTION_BLOCK

// FBs/Components/PrintAndApplyFB
FUNCTION_BLOCK PrintAndApplyFB EXTENDS BaseComponentFB IMPLEMENTS IComponentStatus
VAR_INPUT
	baggerFaulted : BOOL;
	baggerInCycle : BOOL;
	bypass : BOOL;
	dataReady : BOOL;
	LOTAR : BOOL;
	faultInput : BOOL;
	PACycleComplete : BOOL;
	applicatorHome : BOOL;
	heartbeat : BOOL;
	productSensor : BOOL;
	exitConveyorRunAfterPASetting : REAL;
	waitForPrinterFaultSetting : REAL;
END_VAR
VAR_OUTPUT
	state : PRINT_AND_APPLY_STATES;
	commFail : BOOL;
	faultedStatus : BOOL;
	printerNotReady : BOOL;
	printerReadyToApply : BOOL;
	waitingForPrinter : BOOL;
	triggerOutput : BOOL;
	resetOutput : BOOL;
	inhibitCycle : BOOL;
	inhibitConveyor : BOOL;
	runConveyorAfterApply : BOOL;
	waitForPrintFault : BOOL;
	jammedFault : BOOL;
END_VAR
VAR
	resetOutputTimer : MonostableMultivibratorFB();
	exitConveyorRunAfterPA : DelayDwellFB() := (Dwellsetting := 3000);
	inCycleONS : FB_ONS;
	baggerFaultedONS : FB_ONS;
	faultedStatusONS : FB_ONS;
	_beginCycle : BOOL;
	commFailTimer1 : Standard.TON := (PT := T#2S);
	commFailTimer2 : Standard.TON := (PT := T#2S);
	waitForPrinterFaultTimer : Standard.TON;
END_VAR
	
VAR_IN_OUT
END_VAR

//    Function Block: PrintAndApplyFB
//    Description: Statuses and Faults for print and apply
//    Created by: Ben Hess
//    Created Date: December 7th, 2020

// Run parent FB
SUPER^();

printerNotReady := baggerFaulted OR commFail;
waitingForPrinter := (state = PRINT_AND_APPLY_STATES.WaitForLOTAR) OR (state = PRINT_AND_APPLY_STATES.WaitForLabel);


// Timeout on waiting for printer too long
waitForPrinterFaultTimer(IN := waitingForPrinter AND (waitForPrinterFaultSetting > 0) AND enable, 
							PT :=  TO_TIME(waitForPrinterFaultSetting * 1000.0),
							Q=> waitForPrintFault);

//inhibitCycle := (state <> PRINT_AND_APPLY_STATES.Idle) AND enable;
inCycleONS(CLK := baggerInCycle);
baggerFaultedONS(CLK := baggerFaulted);
faultedStatusONS(CLK := faultedStatus);
// Send reset output pulse
resetOutputTimer.DwellSetting := 500;
resetOutputTimer(Q => resetOutput);

exitConveyorRunAfterPA.DwellSetting := TO_DINT(exitConveyorRunAfterPASetting * 1000.0);
exitConveyorRunAfterPA(Q => runConveyorAfterApply);

IF resetONS.Q THEN
	IF faultInput THEN
		resetOutputTimer.Trigger();
	END_IF
	_beginCycle := FALSE;
	exitConveyorRunAfterPA.Reset();
	state := PRINT_AND_APPLY_STATES.Idle;
END_IF
IF NOT enable OR commFail OR faultedStatusONS.OSR OR baggerFaultedONS.OSR THEN
	state := PRINT_AND_APPLY_STATES.Fault;
END_IF

CASE state OF
		
	PRINT_AND_APPLY_STATES.Idle:			//  
											triggerOutput := FALSE;
											inhibitConveyor := FALSE;
											inhibitCycle := FALSE;
											IF _beginCycle THEN
												_beginCycle := FALSE;
												IF dataReady THEN
													state := PRINT_AND_APPLY_STATES.WaitForLOTAR;
												ELSIF LOTAR THEN
													state := PRINT_AND_APPLY_STATES.ReadyToApply;
												ELSE
													state := PRINT_AND_APPLY_STATES.WaitForLabel;
												END_IF
											END_IF
	
	
	PRINT_AND_APPLY_STATES.WaitForLabel:	//  
											IF dataReady OR LOTAR THEN
												state := PRINT_AND_APPLY_STATES.WaitForLOTAR;
											END_IF
											IF productSensor THEN
												inhibitConveyor := TRUE;
											END_IF
											
											inhibitCycle := TRUE;
											
	PRINT_AND_APPLY_STATES.WaitForLOTAR:	//
											IF LOTAR THEN
												state := PRINT_AND_APPLY_STATES.ReadyToApply;
											END_IF
											IF productSensor THEN
												inhibitConveyor := TRUE;
											END_IF
											inhibitCycle := TRUE;
	
	PRINT_AND_APPLY_STATES.ReadyToApply:	//
											inhibitConveyor := FALSE;
											inhibitCycle := FALSE;
											IF productSensor THEN
												exitConveyorRunAfterPA.Trigger();
												triggerOutput := TRUE;
												state := PRINT_AND_APPLY_STATES.Applying;
											END_IF
											
											
	
	PRINT_AND_APPLY_STATES.Applying:		//
											inhibitCycle := FALSE;
											IF NOT productSensor THEN
												triggerOutput := FALSE;
												state := PRINT_AND_APPLY_STATES.Idle;
											END_IF
										
	PRINT_AND_APPLY_STATES.Fault:			//
											triggerOutput := FALSE;
											inhibitConveyor := FALSE;
											inhibitCycle := FALSE;
											exitConveyorRunAfterPA.Reset();
	

END_CASE

printerReadyToApply := state = PRINT_AND_APPLY_STATES.ReadyToApply;

// Comms heartbeat for comm fail fault
commFailTimer1(IN := enable AND heartbeat);
commFailTimer2(IN := enable AND NOT heartbeat);
commFail := commFailTimer1.Q OR commFailTimer2.Q;

// Faulted status from Print and Apply
faultedStatus := NOT commFail AND NOT iPAFaulted AND enable;

METHOD BeginCycle : BOOL
VAR_INPUT
END_VAR
_beginCycle := TRUE;
END_METHOD

METHOD Reset : BOOL
VAR_INPUT
END_VAR
SUPER^.Reset();
END_METHOD

PROPERTY Ready : BOOL
GET
Ready := _ready;
END_GET
SET
_ready := Ready;
END_SET
END_PROPERTY

PROPERTY Mode : DEVICE_MODES
SET
_mode := Mode;
END_SET
GET
Mode := _mode;
END_GET
END_PROPERTY

END_FUNCTION_BLOCK

// FBs/FB_EIPCommsConfigure
FUNCTION_BLOCK FB_EIPCommsConfigure
VAR_INPUT
	rootEIPNode : DED.INode;
	enableWord : DWORD;
END_VAR
VAR
	reconfig : DED.Reconfigure;
	testEnable : BOOL;
	
	tempComapareWord : DWORD;
	_recongfigCommand : BOOL;
	state : INT;
END_VAR

VAR_OUTPUT
	
END_VAR

//    Program: FB_EIPCommsConfigure
//    Description: Allows configuration of individual EIP in in the device tree (enable/disable) 
//    For example, to turn off the comms to a Keyence BCV if it isn't installed
//    Created by: Ben Hess
//    CretestEnableated Date: Wednesday January 6th, 2021

enableWord.0 := Cube67_BN_E_V2.Enable;
enableWord.1 := FestoManifold.Enable;
enableWord.2 := MSFMotor.Enable;
enableWord.3 := Bag_Delivery_EIP_Motor.Enable;
enableWord.4 := Bag_Delivery_Rear_Motor.Enable;
enableWord.5 := Keyence_BCV.Enable;
enableWord.6 := Infeed_Conveyor_IO.Enable;
enableWord.7 := Panther_PA.Enable;
enableWord.8 := IBD_Motor.Enable;

CASE state OF
	
	0:  reconfig.xExecute := FALSE;
		IF enableWord <> tempComapareWord OR _recongfigCommand THEN
			_recongfigCommand := FALSE;
			tempComapareWord := enableWord;
			state := 10;
		END_IF
	
	10:	reconfig.xExecute := TRUE;
		state := 11;
	
	11:	
		IF reconfig.xDone OR reconfig.xError THEN
			state := 0;
		END_IF
	
	
END_CASE




reconfig(
	xExecute:= , 
	xDone=> , 
	xBusy=> , 
	xError=> , 
	itfNode:= rootEIPNode, 
	eError=> );

METHOD ManualReconfig : BOOL
VAR_INPUT
END_VAR
_recongfigCommand := TRUE;
END_METHOD

END_FUNCTION_BLOCK

// Project Information/GetVersion
// This function has been automatically generated from the project information.
{attribute 'signature_flag' := '1073741824'}
{attribute 'register_in_runtime'}
FUNCTION GetVersion : VERSION
VAR_INPUT
	
END_VAR

GetVersion.uiMajor := 0;
GetVersion.uiMinor := 9;
GetVersion.uiServicePack := 15;
GetVersion.uiPatch := 0;

END_FUNCTION

// Project Information/GetTextProperty
// This function has been automatically generated from the project information.
{attribute 'signature_flag' := '1073741824'}
{attribute 'register_in_runtime'}
FUNCTION GetTextProperty : WSTRING
VAR_INPUT
	stKey: WSTRING;
END_VAR

IF stKey = "Author" THEN
	GetTextProperty := "Ben Hess";
ELSIF stKey = "Company" THEN
	GetTextProperty := "Sharp Packaging";
ELSIF stKey = "CompiledLibraryCompatibilityVersion" THEN
	GetTextProperty := "CODESYS V3.5 SP16";
ELSIF stKey = "Project" THEN
	GetTextProperty := "AlphaController";
ELSIF stKey = "Title" THEN
	GetTextProperty := "MOAB Prototype";
ELSIF stKey = "VersionPostfix" THEN
	GetTextProperty := "-alpha/feature/ezfeed";
ELSE
	GetTextProperty := "";
END_IF

END_FUNCTION

// ElectricMachine/Application/Event Handlers/StartDone
FUNCTION StartDone : DWORD
VAR_IN_OUT
	EventPrm: CmpApp.EVTPARAM_CmpApp;
END_VAR
VAR
END_VAR

Globals.firstScan := TRUE;
RecallValues();

END_FUNCTION

// Pro18_1174/Application/Event Handlers/StartDone
FUNCTION StartDone : DWORD
VAR_IN_OUT
	EventPrm: CmpApp.EVTPARAM_CmpApp;
END_VAR
VAR
END_VAR

Globals.firstScan := TRUE;
RecallValues();

END_FUNCTION

// ElectricMachine/Application/Programs/PRG_MainProgram
PROGRAM PRG_MainProgram
VAR
    incrementSolenoidCounter1 : R_TRIG();
    incrementSolenoidCounter2 : R_TRIG();
    incrementSolenoidFailedCounter2 : R_TRIG();
    GripperCycleCount : DINT; //Gripper Cycle Counter
    runPrinterPB : BOOL;
    cycleTimeMax : TIME;
    cycleTimeMaxDINT : DINT;
    ctfb : OSCAT_BASIC.CYCLE_TIME();
    profileThis :BOOL;
    solenoidState1 : SOLENOID_TEST_STATES;
    solenoidState2 : SOLENOID_TEST_STATES;
    getTimeTilPMMI : TimeLeftFB();
	displayPassthroughChangeDistance : REAL;
	displayPassthroughChangeDistance2 : REAL;
	checkSolenoid2ExtendTimer : TON := (PT := T#100MS);
	checkedSolenoid2Status : BOOL;
	firstScanDone : BOOL;
	printDeltaTimer : TON := (PT := T#5S);
	lastPrinterDelta : TIME;
	endPrintOSF : Standard.R_TRIG;
	//CSVWriter : FB_WriteToFile() := (xFilePath := 'C:/printerDelta.csv');
	stringToLog : STRING;
	testWrite : BOOL;
	hmiLight : FB_HMILight;
	versionInfo : VERSION;
	recipieManager : Recipe_Management.RecipeManCommands;
	recipeName : STRING;
	recResult : DWORD;
	testRead : BOOL;
	testCreate : BOOL;
	saveParametersTimer : Standard.TON := (PT := T#10M);
END_VAR

//    Program: Main (PLC_PRG)
//    Description: This program serves as a base for the MOAB Prototype
//    Created by: Ben Hess
//    Created Date: January 16th, 2018

printDeltaTimer(IN := oPrinterStartPrint);
saveParametersTimer(IN := NOT saveParametersTimer.Q AND HMIData.bagsMade.count <> 0);
IF saveParametersTimer.Q THEN
	recResult := recipieManager.GetRecipeNames('Recipes', ADR(recipeName),1,0);
	recResult := recipieManager.ReadAndSaveRecipe(RecipeDefinitionName := 'Recipes', RecipeName := recipeName);
	saveParametersTimer.IN := FALSE;
END_IF

IF testCreate THEN
// 	recResult := recipieManager.CreateRecipe(RecipeDefinitionName := 'Recipes', RecipeName := 'Automatic');
// 	recResult := recipieManager.ReadAndSaveRecipe(RecipeDefinitionName := 'Recipes', RecipeName := recipeName);
 	testCreate := FALSE;
	SaveValues();
END_IF

IF testRead THEN
// 	recResult := recipieManager.GetRecipeNames('Recipes', ADR(recipeName),1,0);
// 	recResult := recipieManager.LoadAndWriteRecipe(RecipeDefinitionName := 'Recipes', RecipeName := recipeName);
 	testRead := FALSE;
	RecallValues();
END_IF

// 
// CSVWriter(
// 	xFilePath:= , 
// 	xText_Write:= , 
// 	xAppend_OverWrite:= TRUE, 
// 	xAppend_Pos:= , 
// 	xWrite:= , 
// 	xRead:= , 
// 	xLine_No_To_Read:= , 
// 	xText_Read=> , 
// 	xDone=> );
// IF CSVWriter.xDone THEN
// 	CSVWriter.xWrite := FALSE;
// END_IF

ctfb(ct_max => cycleTimeMax);
cycleTimeMaxDINT := TIME_TO_DINT(cycleTimeMax);
profileThis := TIME_TO_DINT(ctfb.ct_last) >= 25;
// Run other programs
//PRG_PneumaticHead();
PRG_Bagger();
Faults();
versionInfo := GetVersion();
HMIData.version := Standard.CONCAT(TO_STRING(versionInfo.uiMajor),'.');
	BPLog.AppendToString(ADR(HMIData.version), CONCAT(TO_STRING(versionInfo.uiMinor),'.'));
	BPLog.AppendToString(ADR(HMIData.version), CONCAT(TO_STRING(versionInfo.uiServicePack),'.'));
	BPLog.AppendToString(ADR(HMIData.version), TO_STRING(versionInfo.uiPatch));
	BPLog.AppendToString(ADR(HMIData.version), TO_STRING(GetTextProperty("VersionPostfix")));
IF NOT firstScanDone THEN
	GlobalObjects.CollectionOfLoggable.RegisterAll(internalLogger := Globals.SystemLog);
	GlobalObjects.CollectionOfInitialzable.InitializeAll();
	firstScanDone := TRUE;
	// After first scan turn off flag set by StartDone system event
	Globals.firstScan := FALSE;	
END_IF

// Start executing objects that implement IExecuteAutomatically 
IF firstScanDone THEN
	GlobalObjects.CollectionOfExecutable.ExecuteAll();
	Globals.SystemLog();
END_IF




IF HMIData.ackAllFaults THEN
	GlobalObjects.CollectionOfActiveFaults.AckAll();
	HMIData.ackAllFaults := FALSE;
END_IF

getTimeTilPMMI(targetDate := DT#2018-10-14-8:0:0);


//First scan flag is set by task handler and reset in main routine here
IF Globals.firstScan THEN
    Globals.firstScan := FALSE;
END_IF

displayPassthroughChangeDistance := (UDINT_TO_REAL(Globals.passthroughChangeDistance) / 10);
displayPassthroughChangeDistance2 := (UDINT_TO_REAL(Globals.passthroughChangeDistance2) / 10.0);

END_PROGRAM

// FBs/TimeLeftFB
FUNCTION_BLOCK TimeLeftFB
VAR_INPUT
    targetDate : DATE_AND_TIME;
END_VAR
VAR_OUTPUT
    timeLeft : DATE_AND_TIME;
    
    targetMonths : UINT;
    targetDays : UINT;
    targetHours : UINT;
    targetMinutes : UINT;
    targetSeconds : UINT;
    currentMonths : UINT;
    currentDays : UINT;
    currentHours : UINT;
    currentMinutes : UINT;
    currentSeconds : UINT;
    timeLeftMonths : UINT;
    timeLeftDays : UINT;
    timeLeftHours : UINT;
    timeLeftMinutes : UINT;
    timeLeftSeconds : UINT;
    timeLeftString : STRING[250];
END_VAR
VAR
    iState                    : INT;
    udiUtcTime             : UDINT;
    udiUtcTimeLocal     : UDINT;
    strTimeDate         : SYSTIMEDATE;
    strTimeDateLocal     : SYSTIMEDATE;
    dtDateTimeUTC        : DATE_AND_TIME;
    timeLeftTime        : TIME;
    timeLeftDWORD        : DWORD;
    dDateUTC            : DATE;
    todTimeOfDayUTC        : TOD;
    
    tSysStartTime        : TIME;
    systimeStartNano    : SYSTIME;
    udiStartTimeResult    : UDINT;
    
    udiResult             : UDINT;
    
    
    GetDateAndTime            : DTU.GetDateAndTime;
    SetTimeZoneInformation    : DTU.SetTimeZoneInformation;
    
    dtCurrent                : DATE_AND_TIME;
    dtConcated                : DATE_AND_TIME;
    eWeekday                 : RTCLK.WEEKDAY;
    uiYear                     : UINT;
    uiMonth                     : UINT;
    uiDay                     : UINT;
    uiHour                     : UINT;
    uiMinute                 : UINT;
    uiSecond                 : UINT;
        
    dtuError                : DTU.ERROR;
END_VAR

CASE iState OF

    0:    
        iState:= 1;
        
    1:  // retrieves the target date and time, including the timezone information which was set before
        GetDateAndTime( xExecute:= TRUE);
        IF GetDateAndTime.xDone THEN
            dtCurrent:= GetDateAndTime.dtDateAndTime;
            GetDateAndTime(xExecute:= FALSE);
            //timeLeft := TIME_TO_DT(DT_TO_TIME(targetDate) - DT_TO_TIME(dttarget));
            iState:= 2;
        END_IF
        IF GetDateAndTime.xError THEN
            GetDateAndTime(xExecute:= FALSE);
            iState:= 32767;
        END_IF
    
    2: (*set a spedific date and time --> returns a variable of type DATE_AND_TIME 
         DateConcat --> set only date information --> returns a variable of type DATE
         TODConcat  --> set only the time information  --> returns a variable of TOD (Time of day) *)
        dtConcated := DTU.DTConcat(uiYear:= 2010, uiMonth:= 10, uiDay:= 5, 
                            uiHour:= 9, uiMinute:= 20, uiSecond:= 12, peError:=ADR(dtuError));
        IF dtuError = 0 THEN
            iState := 3;
        ELSE
            iState := 32767;
        END_IF
        
    3:  (*a DATE_AND_TIME variable is splitted in its parts, like year, month, day etc.
            DateSplit --> the same function for a DATE variable
            TODSplit  --> the same function for a TOD variable *)
        dtuError := DTU.DTSplit(
            dtDateAndTime := dtCurrent,
            puiYear := ADR(uiYear), 
            puiMonth := ADR(currentMonths), 
            puiDay := ADR(currentDays), 
            puiHour := ADR(currentHours), 
            puiMinute := ADR(currentMinutes), 
            puiSecond := ADR(currentSeconds));
        dtuError := DTU.DTSplit(
            dtDateAndTime := targetDate,
            puiYear := ADR(uiYear), 
            puiMonth := ADR(targetMonths), 
            puiDay := ADR(targetDays), 
            puiHour := ADR(targetHours), 
            puiMinute := ADR(targetMinutes), 
            puiSecond := ADR(targetSeconds));
            
        IF dtuError = 0 THEN
            iState:= 1;
        ELSE
            iState:= 32767;
        END_IF
        
    32767: ; //error

END_CASE

timeLeftMonths := currentMonths - targetMonths;
timeLeftDays := currentDays - targetDays;
timeLeftHours := currentHours - targetHours;
timeLeftMinutes := currentMinutes - targetMinutes;
timeLeftSeconds := currentSeconds - targetSeconds;

timeLeftString := CONCAT('Time left to PMMI: ', UINT_TO_STRING(timeLeftMonths));
timeLeftString := CONCAT(' Months, ', UINT_TO_STRING(timeLeftDays));
timeLeftString := CONCAT(' Days, ', UINT_TO_STRING(timeLeftHours));
timeLeftString := CONCAT(' Hours, ', UINT_TO_STRING(timeLeftMinutes));
timeLeftString := CONCAT(' Minutes, ', UINT_TO_STRING(timeLeftSeconds));
timeLeftString := CONCAT(' Seconds', '');

timeLeftDWORD := DT_TO_DWORD(targetDate) - DT_TO_DWORD(dtCurrent);
timeLeftDays := DWORD_TO_UINT(timeLeftDWORD / 86000);

END_FUNCTION_BLOCK

// FBs/FB_WriteToFile
FUNCTION_BLOCK FB_WriteToFile
VAR_INPUT
   xFilePath: STRING;
   xText_Write: STRING(2000);
   xAppend_OverWrite: BOOL;
   xAppend_Pos: UDINT;
   xWrite: BOOL;
   xRead: BOOL;
   xLine_No_To_Read: UDINT;   
END_VAR
VAR_OUTPUT
   xText_Read: STRING(2000);
   xDone: BOOL;
END_VAR
VAR
   
// Write Variables
   xWrite_Trig: R_TRIG;
   xStart_Write: BOOL;
   xNew_Line: STRING(2000);
   
// Read Variables
   xRead_Trig: R_TRIG;
   xStart_Read: BOOL;
   xLine_Read: UDINT;
   
   hFile           : RTS_IEC_HANDLE := RTS_INVALID_HANDLE;
   udiBytesRead    : UDINT;
   udiBytesCopied   : UDINT;
   udiWrite      : UDINT;
   udiFileSize     : UDINT;
   udiPos         : UDINT;

//(* Error Codes *)
   udiPosError          : RTS_IEC_RESULT;
   udiCopyError      : RTS_IEC_RESULT;
   udiDeleteError1      : RTS_IEC_RESULT;
   udiDeleteError2      : RTS_IEC_RESULT;
   udiWriteError1      : RTS_IEC_RESULT;
   udiWriteError2      : RTS_IEC_RESULT;
   udiWriteError3      : RTS_IEC_RESULT;
   udiOpenError1      : RTS_IEC_RESULT;
   udiOpenError2      : RTS_IEC_RESULT;
   udiOpenError3      : RTS_IEC_RESULT;
   udiOpenError4      : RTS_IEC_RESULT;

   udiReadError1   : RTS_IEC_RESULT;
   udiReadError2   : RTS_IEC_RESULT;
   udiReadError3   : RTS_IEC_RESULT;
   udiCloseError1   : RTS_IEC_RESULT;
   udiCloseError2   : RTS_IEC_RESULT;
   udiCloseError3   : RTS_IEC_RESULT;
   udiCloseError4   : RTS_IEC_RESULT;
   udiSizeError : RTS_IEC_RESULT;
   udiDirDeleteError: UDINT; 
   udiCreateError: UDINT;
END_VAR

xWrite_Trig();
//xWrite_Trig.PT:= T#500MS;
xWrite_Trig.CLK:= xWrite;
xStart_Write:= xWrite_Trig.Q;

xRead_Trig();
//xRead_Trig.PT:= T#500MS;
xRead_Trig.CLK:= xRead;
xStart_Read:= xRead_Trig.Q;

IF xStart_Write THEN
   xDone:= FALSE;
   IF xAppend_OverWrite THEN 
   hFile:= SysFileOpen(szFile:= xFilePath, am:= ACCESS_MODE.AM_APPEND, pResult:= ADR(udiOpenError1));
   END_IF
   IF xAppend_OverWrite = FALSE THEN
      hFile:= SysFileOpen(szFile:= xFilePath, am:= ACCESS_MODE.AM_WRITE_PLUS, pResult:= ADR(udiOpenError1));
   END_IF
   udiPosError:= SysFileGetPos(hFile:= hFile, pulPos:= ADR(udiPos));
   IF hFile <> RTS_INVALID_HANDLE THEN
      xNew_Line:= concat('$n', xText_Write);
      IF udiPos = 16#0 THEN
         udiWrite:= SysFileWrite(hFile:= hFile, pbyBuffer:= ADR(xText_Write), ulSize:= INT_TO_UDINT(LEN(xText_Write)), pResult:= ADR(udiWriteError1));
      ELSE
         udiWrite:= SysFileWrite(hFile:= hFile, pbyBuffer:= ADR(xNew_Line), ulSize:= INT_TO_UDINT(LEN(xNew_Line)), pResult:= ADR(udiWriteError1));
      END_IF
      udiCloseError1:= SysFileClose(hFile:= hFile);
   END_IF
   xDone:= TRUE;
END_IF

IF xStart_Read THEN
   xDone:= FALSE;
   hFile:= SysFileOpen(szFile:= xFilePath, am:= ACCESS_MODE.AM_READ, pResult:= ADR(udiOpenError1));
   IF hFile <> RTS_INVALID_HANDLE THEN
      udiBytesRead := SysFileRead(hFile:= hFile, pbyBuffer:= ADR(xText_Read), ulSize:=SIZEOF(xText_Read), pResult:=ADR(udiReadError1));
      xText_Read[udiBytesRead]:= 0;
   END_IF
   //xDone:= TRUE;   
END_IF

END_FUNCTION_BLOCK

// FBs/Cylinders/FB_CylinderWithFeedback
FUNCTION_BLOCK FB_CylinderWithFeedback EXTENDS FB_Cylinder IMPLEMENTS ICylinder, IFault
VAR_INPUT
    extendedFeedbackInput : BOOL;    //Extended feedback input from I/O
    retractedFeedbackInput : BOOL;    //Retracted feedback input from I/O
    extendFaultDelay : INT := 1000;        //Extend fault delay in MS
    retractFaultDelay : INT := 1000;        //Retract fault delay in MS
    faultMonitoring : BOOL;                    //Fault monitoring enabled if true
END_VAR
VAR_OUTPUT
    failedToExtend : FB_Fault;            //Failed to Extend Fault
    failedToRetract : FB_Fault;            //Failed to Retract Fault
END_VAR
VAR
    faultIndication : BOOL;            //Overall fault status of cylinder
    extendFaultTimer : TON;            //Extend Fault Timer
    retractFaultTimer : TON;        //Retract Fault Timer
    resetFaults : BOOL;                //Reset faults
END_VAR

METHOD Execute
//This code monitors the positon of the cylinder and raises a fault if the cylinder doesn't reach its
//desired postion within the specified time.

//Initialize timers
extendFaultTimer(PT := INT_TO_TIME(extendFaultDelay));
retractFaultTimer(PT := INT_TO_TIME(retractFaultDelay));

//Only enable timers if we are to be monitoring faults
IF faultMonitoring THEN
    extendFaultTimer.IN := (extendOutput AND NOT extendedFeedbackInput);
    retractFaultTimer.IN := (retractOutput AND NOT retractedFeedbackInput);
ELSE 
        extendFaultTimer.IN := FALSE;
        retractFaultTimer.IN := FALSE;
END_IF

//Rasie the alarms
failedToExtend.faultTrigger := extendFaultTimer.Q;
failedToRetract.faultTrigger := retractFaultTimer.Q;

//Set overall fault indication
//faultIndication := failedToExtend.Active OR failedToRetract;
END_METHOD

END_FUNCTION_BLOCK

// ElectricMachine/Application/PrepareShutdown
FUNCTION PrepareShutdown : DWORD
VAR_IN_OUT
	EventPrm: Component_Manager.EVTPARAM_CmpMgr_Shutdown;
END_VAR
VAR
END_VAR

SaveValues();

END_FUNCTION

// Pro18_1174/Application/Event Handlers/PrepareShutdown
FUNCTION PrepareShutdown : DWORD
VAR_IN_OUT
	EventPrm: Component_Manager.EVTPARAM_CmpMgr_Shutdown;
END_VAR
VAR
END_VAR

SaveValues();

END_FUNCTION

// FBs/Fault/FB_GetTime
FUNCTION_BLOCK FB_GetTime
VAR_INPUT
END_VAR
VAR_OUTPUT
    currentDateAndTime : DATE_AND_TIME;
    
END_VAR
VAR
    iState                    : INT;
    udiUtcTime             : UDINT;
    udiUtcTimeLocal     : UDINT;
    strTimeDate         : SYSTIMEDATE;
    strTimeDateLocal     : SYSTIMEDATE;
    dtDateTimeUTC        : DATE_AND_TIME;
    timeLeftTime        : TIME;
    timeLeftDWORD        : DWORD;
    dDateUTC            : DATE;
    todTimeOfDayUTC        : TOD;
    
    tSysStartTime        : TIME;
    systimeStartNano    : SYSTIME;
    udiStartTimeResult    : UDINT;
    
    udiResult             : UDINT;
    
    
    GetDateAndTime            : DTU.GetDateAndTime;
    SetTimeZoneInformation    : DTU.SetTimeZoneInformation;
    
    dtCurrent                : DATE_AND_TIME;
    dtConcated                : DATE_AND_TIME;
    eWeekday                 : RTCLK.WEEKDAY;
    uiYear                     : UINT;
    uiMonth                     : UINT;
    uiDay                     : UINT;
    uiHour                     : UINT;
    uiMinute                 : UINT;
    uiSecond                 : UINT;
        
    dtuError                : DTU.ERROR;
END_VAR

CASE iState OF

    0:    
        iState:= 1;
        
    1:  // retrieves the target date and time, including the timezone information which was set before
        GetDateAndTime( xExecute:= TRUE);
        IF GetDateAndTime.xDone THEN
            dtCurrent:= GetDateAndTime.dtDateAndTime;
            GetDateAndTime(xExecute:= FALSE);
			currentDateAndTime := dtCurrent;
            //timeLeft := TIME_TO_DT(DT_TO_TIME(targetDate) - DT_TO_TIME(dttarget));
            iState:= 2;
        END_IF
        IF GetDateAndTime.xError THEN
            GetDateAndTime(xExecute:= FALSE);
            iState:= 32767;
        END_IF
    
    2: (*set a spedific date and time --> returns a variable of type DATE_AND_TIME 
         DateConcat --> set only date information --> returns a variable of type DATE
         TODConcat  --> set only the time information  --> returns a variable of TOD (Time of day) *)
        IF dtuError = 0 THEN
            iState := 3;
        ELSE
            iState := 32767;
        END_IF
        
    3:  (*a DATE_AND_TIME variable is splitted in its parts, like year, month, day etc.
            DateSplit --> the same function for a DATE variable
            TODSplit  --> the same function for a TOD variable *)

            
        IF dtuError = 0 THEN
            iState:= 1;
        ELSE
            iState:= 32767;
        END_IF
        
    32767: ; //error

END_CASE

END_FUNCTION_BLOCK

// ObjectHandling/FB_CollectionHandlerAll
FUNCTION_BLOCK FINAL FB_CollectionHandlerAll
VAR_INPUT
END_VAR
VAR
	Collection: ARRAY[0..GlobalObjects.MAX_OBJECTS] OF IAllObjects; // object array
	ObjNames   : ARRAY[0..GlobalObjects.MAX_OBJECTS] OF STRING;
	_ArrayOver   : BOOL;
	_BadObj      : INT;
	_DupeObj   : INT;
	_OverObj   : INT;
	_TotalObj   : UINT;
END_VAR

METHOD FINAL AddObject
VAR_INPUT
	Obj   : IAllObjects;
END_VAR
VAR
	AnyObject : IAllObjects;
	Fault : IFault;
	Cylinder : ICylinder;
	PositionableMotor : IPositionableMotor;
	Logger : IMachineLogger;
	Loggable : ILoggable;
	Executable : IExecuteAutomatically;
	Initializable : IInitializable;
	J   : UINT;
END_VAR
IF (__QUERYINTERFACE(Obj, AnyObject)) THEN
   // make sure haven't already added this object
   FOR J:= 1 TO _TotalObj DO
      IF Collection[J] = AnyObject THEN
         // object pointer matches - dupe!
         _DupeObj:= _DupeObj + 1;
         RETURN;
      END_IF
   END_FOR
   
   IF _TotalObj < GlobalObjects.MAX_OBJECTS THEN
      Collection[_TotalObj]:= AnyObject;
      ObjNames[_TotalObj]:= Obj.InstanceName;
	   _TotalObj:= _TotalObj + 1;
   ELSE
      _ArrayOver:= TRUE;
      _OverObj:= _OverObj + 1;
   END_IF
ELSE
   _BadObj:= _BadObj + 1;
END_IF

// Add object to proper collection based on its interfaces
IF (__QUERYINTERFACE(Obj, Fault)) THEN
	GlobalObjects.CollectionOfFaults.AddObject(Fault);
END_IF

// IF (__QUERYINTERFACE(Obj, Cylinder)) THEN
// 	GlobalObjects.CollectionOfCylinders.AddObject(Cylinder);
// END_IF
// 
// IF (__QUERYINTERFACE(Obj, PositionableMotor)) THEN
// 	GlobalObjects.CollectionOfPositionableMotors.AddObject(PositionableMotor);
// END_IF

IF (__QUERYINTERFACE(Obj, Logger)) THEN
	GlobalObjects.CollectionOfLogs.AddObject(Logger);
END_IF

IF (__QUERYINTERFACE(Obj, Loggable)) THEN
	GlobalObjects.CollectionOfLoggable.AddObject(Loggable);
END_IF

IF (__QUERYINTERFACE(Obj, Executable)) THEN
	GlobalObjects.CollectionOfExecutable.AddObject(Executable);
END_IF

IF (__QUERYINTERFACE(Obj, Initializable)) THEN
	GlobalObjects.CollectionOfInitialzable.AddObject(Initializable);
END_IF
END_METHOD

END_FUNCTION_BLOCK

// FBs/Components/BagDeliveryFB_BothMotors
FUNCTION_BLOCK BagDeliveryFB_BothMotors EXTENDS BaseComponentFB IMPLEMENTS IComponentStatus
VAR_INPUT
    feedBagPB : BOOL;                // Manually Feed bag out
	jogForwardPB : BOOL;
	jogReversePB : BOOL;
    bagsToFeedSetpoint : INT;        // Bags to feed setpoint for testing
    reverseDistanceSetpoint : REAL := -3;  // Distance to reverse
    bagLengthSetpoint : REAL := 23.5;  // Bag length to feed
    accelSetpoint : INT := 600;            // Acceleration Setpoint
    decelSetpoint : INT := 2000;        // Deceleration Setpoint
    reverseVelocitySetpoint : INT := 3;            // Reverse Velocity setoint (IPS)
    feedVelocitySetpoint : INT := 55;            // Bag Feed Velocity setoint (IPS)
    printVelocitySetpoint : UDINT := 6;            // Print speed (IPS)
    sealOffsetSetpoint : REAL := 1.5;            // Seal Offset
    printOffsetSetpoint : REAL := 3;            // Print Offset
    printLengthSetpoint : REAL := 8;                    // Print length
	reverseToPrintHeadSetpoint : REAL := -1.25;
	feedToPhotoeyeSetpoint : REAL := 2.0;
	useLastPrinterDelta : BOOL := TRUE;
	tensionFailONS : FB_ONS;
END_VAR
VAR_OUTPUT
    state : BAG_DELIVERY_STATES;    // Current state of bag delivery component
	reverseFault : FB_Fault(name := 'Reverse Fault');
	noBagOverEye : FB_Fault(name := 'No bag over Photoeye');
	bagTensionFault : FB_Fault(name := 'Bag Tension Fault');
END_VAR
VAR
    delay : TON := (PT := T#100MS);    // Delay for testing
	jogForwardONS: FB_ONS;
	jogReverseONS: FB_ONS;
	delayForReverseFault : Standard.TON;
	autoFeedDelay : TON := (PT := T#200MS);
	sealBarToPrintHeadLength : REAL;
    bagsCurrentlyFed  :INT;            // Bags currently fed for testing
    remainingLength : REAL;            // Remaining bag length after print
	delayForPrintFeed : TIME := T#250MS;
	printerExtraFeedLength : REAL := 0.25;
    //bagFeedMasterMotor : FB_AppliedMotionStepServoTCP();
    //bagFeedMasterMotor : FB_AppliedMotionBagDeliveryMotor();
	bagFeedMasterMotor : FB_AppliedMotionBagDeliveryMotor_1();
	//bagFeedRearMotor : FB_AppliedMotionBagDeliveryMotor_1();
	bagFeedRearMotor : FB_AppliedMotionStepServoEIPBase();
	accelPercent : REAL := 0.1;
	decelPercent : REAL := 0.05;
    _amReverseBag : BOOL;            // Auto Mode - Reverse bag
    _amFeedBagOut : BOOL;            // Auto Mode - Feed new bag out
    _amWaitForPrinter : BOOL;        // Auto Mode - wait for printer
    _amPrinterReady : BOOL;            // Auto Mode - Printer is ready
    _amStartPrint : BOOL;            // Auto Mode - Start Printing
    _amPrinterDone : BOOL;             // Auto Mode - Printer is Done
	_amFeedToEye : BOOL;			  // Auto Mode - Feed Bag to Eye
END_VAR

//    Function Block: BagDeliveryFB
//    Description: This is the state machine for the bag delivery test rig
//    
//    Created by: Ben Hess
//    Created Date: Thursday, April 19, 2018

SUPER^();
tensionFailONS(CLK := iBagTensionFault);

delay();
delayForReverseFault();
autoFeedDelay(IN := _amFeedBagOut);
// This is the master Applied Motion motor
IF useLastPrinterDelta THEN
	IF Globals.lastPrinterDelta >= T#90MS THEN
		delayForPrintFeed := Globals.lastPrinterDelta - T#80MS;
	ELSE
		delayForPrintFeed := T#10MS;
	END_IF
END_IF
bagLengthSetpoint := HMIData.bagLength;
printVelocitySetpoint := HMIData.printSpeed;
sealOffsetSetpoint := HMIData.bagSkirtLength;
printOffsetSetpoint := HMIData.printOffset;
sealBarToPrintHeadLength := ABS(reverseToPrintHeadSetpoint) + 2.25;
printLengthSetpoint := HMIData.printLength;
reverseVelocitySetpoint := TO_INT(HMIData.bagReverseSpeed);
feedVelocitySetpoint := TO_INT(HMIData.bagForwardSpeed);

(*bagFeedMasterMotor(modbusInputParameters := BagDeliverMasterMotorModbusInputs, 
                    stepsPerInchSetpoint := Globals.STEPS_PER_INCH_20_DEGREE_BAG_DELIVERY, 
                    reversePolarity := FALSE, 
                    slave := Bag_Delivery_Master_Motor);*)
bagFeedMasterMotor(ptrEIPInputs := ADR(bagDeliveryMotorInputs),
                ptrEIPOutputs := ADR(bagDeliveryMotorOutputs),
                stepsPerInchSetpoint := Globals.STEPS_PER_INCH_20_DEGREE_BAG_DELIVERY,
                //faultHandler := PRG_Bagger.faultHandler,
				reversePolarity := FALSE, 
				defaultCurrentSetpoint := 1150, 
				commFail := Bag_Delivery_EIP_Motor.eState <> IoDrvEthernetIP.AdapterState.RUNNING);
bagFeedMasterMotor.Execute();

bagFeedRearMotor(ptrEIPInputs := ADR(bagRearMotorInputs),
                ptrEIPOutputs := ADR(bagRearMotorOutputs),
                stepsPerInchSetpoint := Globals.STEPS_PER_INCH_20_DEGREE_BAG_DELIVERY,
                //faultHandler := PRG_Bagger.faultHandler,
				reversePolarity := FALSE, 
				defaultCurrentSetpoint := 1150, 
				commFail := Bag_Delivery_Rear_Motor.eState <> IoDrvEthernetIP.AdapterState.RUNNING);
bagFeedRearMotor.Execute();

IF enableONS.Q OR resetONS.Q THEN
    IF _mode = DEVICE_MODES.Manual THEN 
        state := BAG_DELIVERY_STATES.Manual;
    ELSE
        state := BAG_DELIVERY_STATES.Idle;
    END_IF
	_reset := FALSE;
	ClearCommands();
END_IF
jogForwardONS(CLK := jogForwardPB);
jogReverseONS(CLK := jogReversePB);
IF NOT enable THEN
    state := BAG_DELIVERY_STATES.Idle;
END_IF
delay();
_ready := (_mode = DEVICE_MODES.Auto) AND (NOT (state = BAG_DELIVERY_STATES.Fault) OR NOT (state = BAG_DELIVERY_STATES.Idle));

IF tensionFailONS.OSR THEN
	bagTensionFault.Trigger();
END_IF

CASE state OF
    BAG_DELIVERY_STATES.Idle :                     
													IF _mode = DEVICE_MODES.Manual THEN 
														state := BAG_DELIVERY_STATES.Manual;
													ELSIF NOT iBagNotPresent OR Globals.enableDryCycle THEN
														state := BAG_DELIVERY_STATES.Ready;
													ELSIF iBagNotPresent AND (_amFeedToEye OR _amReverseBag) THEN
														state := BAG_DELIVERY_STATES.FeedToEye;
														_amFeedToEye := FALSE;
													END_IF
													IF jogForwardONS.OSR THEN
														bagFeedMasterMotor.MoveDistance(distance := 30, 
                                                                                    acceleration := accelSetpoint, 
                                                                                    deceleration := decelSetpoint, 
                                                                                    velocity := REAL_TO_INT((1 * Globals.VELOCITY_IPS_MULTIPLIER_20_DEGREE_BAG_DELIVERY)));
														bagFeedRearMotor.MoveDistance(distance := 30, 
                                                                                    acceleration := accelSetpoint, 
                                                                                    deceleration := decelSetpoint, 
                                                                                    velocity := REAL_TO_INT((1 * Globals.VELOCITY_IPS_MULTIPLIER_20_DEGREE_BAG_DELIVERY)));
													ELSIF jogReverseONS.OSR THEN
														bagFeedMasterMotor.MoveDistance(distance := -30, 
                                                                                    acceleration := accelSetpoint, 
                                                                                    deceleration := decelSetpoint, 
                                                                                    velocity := REAL_TO_INT((1 * Globals.VELOCITY_IPS_MULTIPLIER_20_DEGREE_BAG_DELIVERY)));
														bagFeedRearMotor.MoveDistance(distance := -30, 
                                                                                    acceleration := accelSetpoint, 
                                                                                    deceleration := decelSetpoint, 
                                                                                    velocity := REAL_TO_INT((1 * Globals.VELOCITY_IPS_MULTIPLIER_20_DEGREE_BAG_DELIVERY)));
													ELSIF jogForwardONS.OSF OR jogReverseONS.OSF THEN
														bagFeedMasterMotor.Stop();
														bagFeedRearMotor.Stop();
													END_IF
    
	BAG_DELIVERY_STATES.FeedToEye :					//Feed to photoeye if not present
													bagFeedMasterMotor.MoveDistance(distance := feedToPhotoeyeSetpoint, 
                                                                                    acceleration := accelSetpoint, 
                                                                                    deceleration := decelSetpoint, 
                                                                                    velocity := REAL_TO_INT((feedToPhotoeyeSetpoint * Globals.VELOCITY_IPS_MULTIPLIER_20_DEGREE_BAG_DELIVERY)));
													bagFeedRearMotor.MoveDistance(distance := feedToPhotoeyeSetpoint, 
                                                                                    acceleration := accelSetpoint, 
                                                                                    deceleration := decelSetpoint, 
                                                                                    velocity := REAL_TO_INT((feedToPhotoeyeSetpoint * Globals.VELOCITY_IPS_MULTIPLIER_20_DEGREE_BAG_DELIVERY)));
													state := BAG_DELIVERY_STATES.FeedingToEye;
													
	BAG_DELIVERY_STATES.FeedingToEye :				// Stop once photoeye seen
													delay.PT := T#3S;
													delay.IN := TRUE;
													IF NOT iBagNotPresent THEN
														bagFeedMasterMotor.Stop();
														bagFeedRearMotor.Stop();
														state := BAG_DELIVERY_STATES.Idle;
														delay.IN := FALSE;
													END_IF
													IF delay.Q THEN
														state := BAG_DELIVERY_STATES.Fault;
														noBagOverEye.Trigger();
														delay.IN := FALSE;
													END_IF
	
    BAG_DELIVERY_STATES.Reverse :                    // Reverse to break perf
                                                    bagFeedMasterMotor.MoveDistance(distance := reverseDistanceSetpoint, 
                                                                                    acceleration := TO_INT((ABS(reverseDistanceSetpoint) * Globals.STEPS_PER_INCH_20_DEGREE_BAG_DELIVERY) *  accelPercent),
                                                                                    deceleration := TO_INT((ABS(reverseDistanceSetpoint) * Globals.STEPS_PER_INCH_20_DEGREE_BAG_DELIVERY) *  decelPercent), 
                                                                                    velocity := REAL_TO_INT((reverseVelocitySetpoint * Globals.VELOCITY_IPS_MULTIPLIER_20_DEGREE_BAG_DELIVERY)));  
													bagFeedRearMotor.MoveDistance(distance := reverseDistanceSetpoint, 
                                                                                    acceleration := TO_INT((ABS(reverseDistanceSetpoint) * Globals.STEPS_PER_INCH_20_DEGREE_BAG_DELIVERY) *  accelPercent),
                                                                                    deceleration := TO_INT((ABS(reverseDistanceSetpoint) * Globals.STEPS_PER_INCH_20_DEGREE_BAG_DELIVERY) *  decelPercent), 
                                                                                    velocity := REAL_TO_INT((reverseVelocitySetpoint * Globals.VELOCITY_IPS_MULTIPLIER_20_DEGREE_BAG_DELIVERY)));    
                                                        state := BAG_DELIVERY_STATES.Reversing;
                                                    
                                                    
    BAG_DELIVERY_STATES.Reversing :                    // Back up until we see the trailing edge of the bag
														 IF iBagNotPresent OR Globals.enableDryCycle THEN
															delay.PT := T#10MS;
															delay.IN := TRUE;
															IF delay.Q THEN
																bagFeedMasterMotor.Stop();
																bagFeedRearMotor.Stop();
																delay.IN := FALSE;
																delayForReverseFault.IN := FALSE;
																state := BAG_DELIVERY_STATES.ReverseToPrinthead;
															END_IF
														ELSIF bagFeedMasterMotor.CommandAcknowledged AND NOT iBagNotPresent THEN
															delayForReverseFault.PT := T#3000MS;
															delayForReverseFault.IN := TRUE;
															IF delayForReverseFault.Q THEN
																reverseFault.Trigger();
																bagFeedMasterMotor.Stop();
																bagFeedRearMotor.Stop();
															delayForReverseFault.IN := FALSE;
															state := BAG_DELIVERY_STATES.Fault; 
															END_IF
															
														END_IF
											
                                                  
													
	BAG_DELIVERY_STATES.ReverseToPrinthead :                    // Reverse to print head
                                                    bagFeedMasterMotor.MoveDistance(distance := reverseToPrintHeadSetpoint, 
                                                                                    acceleration := TO_INT((ABS(reverseToPrintHeadSetpoint) * Globals.STEPS_PER_INCH_20_DEGREE_BAG_DELIVERY) *  accelPercent),
                                                                                    deceleration := TO_INT((ABS(reverseToPrintHeadSetpoint) * Globals.STEPS_PER_INCH_20_DEGREE_BAG_DELIVERY) *  decelPercent), 
                                                                                    velocity := REAL_TO_INT((reverseVelocitySetpoint * Globals.VELOCITY_IPS_MULTIPLIER_20_DEGREE_BAG_DELIVERY))); 
													bagFeedRearMotor.MoveDistance(distance := reverseToPrintHeadSetpoint, 
                                                                                    acceleration := TO_INT((ABS(reverseToPrintHeadSetpoint) * Globals.STEPS_PER_INCH_20_DEGREE_BAG_DELIVERY) *  accelPercent),
                                                                                    deceleration := TO_INT((ABS(reverseToPrintHeadSetpoint) * Globals.STEPS_PER_INCH_20_DEGREE_BAG_DELIVERY) *  decelPercent), 
                                                                                    velocity := REAL_TO_INT((reverseVelocitySetpoint * Globals.VELOCITY_IPS_MULTIPLIER_20_DEGREE_BAG_DELIVERY)));    
                                                    state := BAG_DELIVERY_STATES.ReversingToPrintHead;
													
	BAG_DELIVERY_STATES.ReversingToPrintHead :                    // Reverse to break perf
                                                   	delay.PT := T#50MS;
													delay.IN := TRUE;
													
													IF delay.Q THEN
														IF bagFeedMasterMotor.CommandAcknowledged AND bagFeedMasterMotor.InPosition THEN
                                                        	state := BAG_DELIVERY_STATES.ReverseDone;
                                                    	END_IF
														delay.IN := FALSE;
													END_IF
                                                    
    BAG_DELIVERY_STATES.ReverseDone :                // We don't print in semi auto or manual mode.  In auto mode if the printer is selected then we move to those states
                                                    IF _mode = DEVICE_MODES.SemiAuto OR _mode = DEVICE_MODES.Manual OR (_mode  = DEVICE_MODES.Auto AND autoFeedDelay.Q) THEN
                                                        IF bagFeedMasterMotor.CommandAcknowledged THEN
															state := BAG_DELIVERY_STATES.FeedBagOut;
                                                        	remainingLength := bagLengthSetpoint;
                                                        	_amFeedBagOut := FALSE;
														END_IF
														
                                                    ELSIF (_mode  = DEVICE_MODES.Auto AND _amWaitForPrinter) THEN
                                                        IF bagFeedMasterMotor.CommandAcknowledged THEN
															state := BAG_DELIVERY_STATES.WaitingForPrinter;
															remainingLength := bagLengthSetpoint - (printLengthSetpoint + printOffsetSetpoint + printerExtraFeedLength);
															_amWaitForPrinter := FALSE;  
														END_IF  
                                                    END_IF
                                                        
                                                    
    BAG_DELIVERY_STATES.WaitingForPrinter :            // 
                                                    IF (_mode  = DEVICE_MODES.Auto AND _amPrinterReady) THEN
														IF printOffsetSetpoint <> 0 THEN
															state := BAG_DELIVERY_STATES.FeedToPrintOffset;
														ELSE
															state := BAG_DELIVERY_STATES.FedToPrintOffset;
														END_IF
                                                        
                                                        _amPrinterReady := FALSE;
                                                    END_IF
                                                        
    BAG_DELIVERY_STATES.FeedToPrintOffset :            // 
                                                    bagFeedMasterMotor.MoveDistance(distance := printOffsetSetpoint, 
                                                                                    acceleration := accelSetpoint, 
                                                                                    deceleration := decelSetpoint, 
                                                                                    velocity := REAL_TO_INT((feedVelocitySetpoint * Globals.VELOCITY_IPS_MULTIPLIER_20_DEGREE_BAG_DELIVERY)));  
													bagFeedRearMotor.MoveDistance(distance := printOffsetSetpoint, 
                                                                                    acceleration := accelSetpoint, 
                                                                                    deceleration := decelSetpoint, 
                                                                                    velocity := REAL_TO_INT((feedVelocitySetpoint * Globals.VELOCITY_IPS_MULTIPLIER_20_DEGREE_BAG_DELIVERY)));  
                                                        state := BAG_DELIVERY_STATES.FeedingToPrintOffset;
                                                    
    BAG_DELIVERY_STATES.FeedingToPrintOffset :        // 
													delay.PT := T#50MS;
													delay.IN := TRUE;
													
													IF delay.Q THEN
														IF bagFeedMasterMotor.CommandAcknowledged AND bagFeedMasterMotor.InPosition THEN
                                                        	state := BAG_DELIVERY_STATES.FedToPrintOffset;
                                                    	END_IF
														delay.IN := FALSE;
													END_IF
                                                    
                                                    
    BAG_DELIVERY_STATES.FedToPrintOffset :            // 
                                                    IF (_mode  = DEVICE_MODES.Auto AND _amStartPrint) THEN
                                                        state := BAG_DELIVERY_STATES.FeedAtPrintSpeed;
                                                        _amStartPrint := FALSE;
                                                    END_IF
                                                    
    BAG_DELIVERY_STATES.FeedAtPrintSpeed :            // 
													delay.PT := delayForPrintFeed;
                                                    delay.IN := TRUE;
													
													IF delay.Q THEN
														bagFeedMasterMotor.MoveDistance(distance := printLengthSetpoint + printerExtraFeedLength, 
                                                                                    acceleration := accelSetpoint, 
                                                                                    deceleration := decelSetpoint, 
                                                                                    velocity := REAL_TO_INT((printVelocitySetpoint * Globals.VELOCITY_IPS_MULTIPLIER_20_DEGREE_BAG_DELIVERY)));  
														bagFeedRearMotor.MoveDistance(distance := printLengthSetpoint + printerExtraFeedLength, 
                                                                                    acceleration := accelSetpoint, 
                                                                                    deceleration := decelSetpoint, 
                                                                                    velocity := REAL_TO_INT((printVelocitySetpoint * Globals.VELOCITY_IPS_MULTIPLIER_20_DEGREE_BAG_DELIVERY)));  
                                                        state := BAG_DELIVERY_STATES.FeedingAtPrintSpeed;
														delay.IN := FALSE;
													END_IF
                                                    
    BAG_DELIVERY_STATES.FeedingAtPrintSpeed :        // 
													delay.PT := T#50MS;
													delay.IN := TRUE;
													IF delay.Q THEN
														IF bagFeedMasterMotor.CommandAcknowledged AND bagFeedMasterMotor.InPosition THEN
                                                        	state := BAG_DELIVERY_STATES.FedAtPrintSpeed;
                                                    	END_IF
														delay.IN := FALSE;
													END_IF
                                                   
                                                    
    BAG_DELIVERY_STATES.FedAtPrintSpeed :            // 
                                                    IF (_mode  = DEVICE_MODES.Auto AND _amPrinterDone) THEN
                                                        state := BAG_DELIVERY_STATES.FeedBagOut;
                                                        _amPrinterDone := FALSE;
                                                    END_IF
                                                    
    BAG_DELIVERY_STATES.FeedBagOut :                // Feed bag length out
                                                    //bagFeedMasterMotor.MoveDistanceFinal(distance := (remainingLength + sealOffsetSetpoint + (reverseToPrintHeadSetpoint*-1)), 
													bagFeedMasterMotor.MoveDistanceFinal(distance := (remainingLength + sealBarToPrintHeadLength) - sealOffsetSetpoint, 
                                                                                        acceleration := accelSetpoint, 
                                                                                        deceleration := decelSetpoint, 
                                                                                        velocity := REAL_TO_INT((feedVelocitySetpoint * Globals.VELOCITY_IPS_MULTIPLIER_20_DEGREE_BAG_DELIVERY)));
													bagFeedRearMotor.MoveDistance(distance := (remainingLength + sealBarToPrintHeadLength) - sealOffsetSetpoint, 
                                                                                        acceleration := accelSetpoint, 
                                                                                        deceleration := decelSetpoint, 
                                                                                        velocity := REAL_TO_INT((feedVelocitySetpoint * Globals.VELOCITY_IPS_MULTIPLIER_20_DEGREE_BAG_DELIVERY)));
                                                    state := BAG_DELIVERY_STATES.FeedingBagOut;    
    
    BAG_DELIVERY_STATES.FeedingBagOut :                // Wait until move is done
													delay.PT := T#50MS;
													delay.IN := TRUE;
													IF delay.Q THEN
														IF bagFeedMasterMotor.CommandAcknowledged AND bagFeedMasterMotor.InPosition THEN
                                                        state := BAG_DELIVERY_STATES.FedBagOut;
														
                                                    	END_IF
														delay.IN := FALSE;
													END_IF
                                                    
    
    BAG_DELIVERY_STATES.FedBagOut :                    // Go to the next ready state
                                                    IF _mode = DEVICE_MODES.Manual THEN 
                                                        state := BAG_DELIVERY_STATES.Manual;
                                                    ELSE
                                                        state := BAG_DELIVERY_STATES.Ready;
                                                    END_IF
													HMIData.driveRollerClean.SetCount(HMIData.driveRollerClean.count + TO_INT(bagLengthSetpoint));
                                                    Globals.bagDeliveryCycleCount := Globals.bagDeliveryCycleCount + 1;
    
